   ELSE
       // ruch czarnych
       // 
       //ruch po skosie 
       #wykonuj_petle := TRUE;
       #poz_temp := #hetman.pozycja;
       WHILE #wykonuj_petle DO
           #poz_temp.x += 1;
           #poz_temp.y += 1;
           IF "sprawdz_czy_na_szachownicy"(#poz_temp) = true THEN
               IF "sprawdz_czy_wolne"(pozycja := #poz_temp, szachownica := #szachownica) = true THEN
                   IF #poz_temp.x = #polozenie_krola.x  AND #poz_temp.y = #polozenie_krola.y  THEN
                       #sprawdz_czy_hetman_szach := true;
                   END_IF;
               ELSIF "sprawdz_czy_zajete"(pozycja := #poz_temp, szachownica := #szachownica) = 2 THEN
                   IF #poz_temp.x = #polozenie_krola.x  AND #poz_temp.y = #polozenie_krola.y  THEN
                       #sprawdz_czy_hetman_szach := true;
                   ELSE
                       #wykonuj_petle := false;
                   END_IF;
               ELSE
                   #wykonuj_petle := false;
               END_IF;
           ELSE
               #wykonuj_petle := false;
           END_IF;
       END_WHILE;
       #wykonuj_petle := TRUE;
       #poz_temp := #hetman.pozycja;
       WHILE #wykonuj_petle DO
           #poz_temp.x += 1;
           #poz_temp.y -= 1;
           IF "sprawdz_czy_na_szachownicy"(#poz_temp) = true THEN
               IF "sprawdz_czy_wolne"(pozycja := #poz_temp, szachownica := #szachownica) = true THEN
                   IF #poz_temp.x = #polozenie_krola.x  AND #poz_temp.y = #polozenie_krola.y  THEN
                       #sprawdz_czy_hetman_szach := true;
                   END_IF;
               ELSIF "sprawdz_czy_zajete"(pozycja := #poz_temp, szachownica := #szachownica) = 2 THEN
                   IF #poz_temp.x = #polozenie_krola.x  AND #poz_temp.y = #polozenie_krola.y  THEN
                       #sprawdz_czy_hetman_szach := true;
                   ELSE
                       #wykonuj_petle := false;
                   END_IF;
               ELSE
                   #wykonuj_petle := false;
               END_IF;
           ELSE
               #wykonuj_petle := false;
           END_IF;
       END_WHILE;
       #wykonuj_petle := TRUE;
       #poz_temp := #hetman.pozycja;
       WHILE #wykonuj_petle DO
           #poz_temp.x -= 1;
           #poz_temp.y += 1;
           IF "sprawdz_czy_na_szachownicy"(#poz_temp) = true THEN
               IF "sprawdz_czy_wolne"(pozycja := #poz_temp, szachownica := #szachownica) = true THEN
                   IF #poz_temp.x = #polozenie_krola.x  AND #poz_temp.y = #polozenie_krola.y  THEN
                       #sprawdz_czy_hetman_szach := true;
                   END_IF;
               ELSIF "sprawdz_czy_zajete"(pozycja := #poz_temp, szachownica := #szachownica) = 2 THEN
                   IF #poz_temp.x = #polozenie_krola.x  AND #poz_temp.y = #polozenie_krola.y  THEN
                       #sprawdz_czy_hetman_szach := true;
                   ELSE
                       #wykonuj_petle := false;
                   END_IF;
               ELSE
                   #wykonuj_petle := false;
               END_IF;
           ELSE
               #wykonuj_petle := false;
           END_IF;
       END_WHILE;
       #wykonuj_petle := TRUE;
       #poz_temp := #hetman.pozycja;
       WHILE #wykonuj_petle DO
           #poz_temp.x -= 1;
           #poz_temp.y -= 1;
           IF "sprawdz_czy_na_szachownicy"(#poz_temp) = true THEN
               IF "sprawdz_czy_wolne"(pozycja := #poz_temp, szachownica := #szachownica) = true THEN
                   IF #poz_temp.x = #polozenie_krola.x  AND #poz_temp.y = #polozenie_krola.y  THEN
                       #sprawdz_czy_hetman_szach := true;
                   END_IF;
               ELSIF "sprawdz_czy_zajete"(pozycja := #poz_temp, szachownica := #szachownica) = 2 THEN
                   IF #poz_temp.x = #polozenie_krola.x  AND #poz_temp.y = #polozenie_krola.y  THEN
                       #sprawdz_czy_hetman_szach := true;
                   ELSE
                       #wykonuj_petle := false;
                   END_IF;
               ELSE
                   #wykonuj_petle := false;
               END_IF;
           ELSE
               #wykonuj_petle := false;
           END_IF;
       END_WHILE;
       //ruch poziomo i pionowo
       #wykonuj_petle := TRUE;
       #poz_temp := #hetman.pozycja;
       WHILE #wykonuj_petle DO
           #poz_temp.x += 1;
           #poz_temp.y += 0;
           IF "sprawdz_czy_na_szachownicy"(#poz_temp) = true THEN
               IF "sprawdz_czy_wolne"(pozycja := #poz_temp, szachownica := #szachownica) = true THEN
                   IF #poz_temp.x = #polozenie_krola.x  AND #poz_temp.y = #polozenie_krola.y  THEN
                       #sprawdz_czy_hetman_szach := true;
                   END_IF;
               ELSIF "sprawdz_czy_zajete"(pozycja := #poz_temp, szachownica := #szachownica) = 2 THEN
                   IF #poz_temp.x = #polozenie_krola.x  AND #poz_temp.y = #polozenie_krola.y  THEN
                       #sprawdz_czy_hetman_szach := true;
                   ELSE
                       #wykonuj_petle := false;
                   END_IF;
               ELSE
                   #wykonuj_petle := false;
               END_IF;
           ELSE
               #wykonuj_petle := false;
           END_IF;
       END_WHILE;
       #wykonuj_petle := TRUE;
       #poz_temp := #hetman.pozycja;
       WHILE #wykonuj_petle DO
           #poz_temp.x += 0;
           #poz_temp.y += 1;
           IF "sprawdz_czy_na_szachownicy"(#poz_temp) = true THEN
               IF "sprawdz_czy_wolne"(pozycja := #poz_temp, szachownica := #szachownica) = true THEN
                   IF #poz_temp.x = #polozenie_krola.x  AND #poz_temp.y = #polozenie_krola.y  THEN
                       #sprawdz_czy_hetman_szach := true;
                   END_IF;
               ELSIF "sprawdz_czy_zajete"(pozycja := #poz_temp, szachownica := #szachownica) = 2 THEN
                   IF #poz_temp.x = #polozenie_krola.x  AND #poz_temp.y = #polozenie_krola.y  THEN
                       #sprawdz_czy_hetman_szach := true;
                   ELSE
                       #wykonuj_petle := false;
                   END_IF;
               ELSE
                   #wykonuj_petle := false;
               END_IF;
           ELSE
               #wykonuj_petle := false;
           END_IF;
       END_WHILE;
       #wykonuj_petle := TRUE;
       #poz_temp := #hetman.pozycja;
       WHILE #wykonuj_petle DO
           #poz_temp.x += -1;
           #poz_temp.y += 0;
           IF "sprawdz_czy_na_szachownicy"(#poz_temp) = true THEN
               IF "sprawdz_czy_wolne"(pozycja := #poz_temp, szachownica := #szachownica) = true THEN
                   IF #poz_temp.x = #polozenie_krola.x  AND #poz_temp.y = #polozenie_krola.y  THEN
                       #sprawdz_czy_hetman_szach := true;
                   END_IF;
               ELSIF "sprawdz_czy_zajete"(pozycja := #poz_temp, szachownica := #szachownica) = 2 THEN
                   IF #poz_temp.x = #polozenie_krola.x  AND #poz_temp.y = #polozenie_krola.y  THEN
                       #sprawdz_czy_hetman_szach := true;
                   ELSE
                       #wykonuj_petle := false;
                   END_IF;
               ELSE
                   #wykonuj_petle := false;
               END_IF;
           ELSE
               #wykonuj_petle := false;
           END_IF;
       END_WHILE;
       #wykonuj_petle := TRUE;
       #poz_temp := #hetman.pozycja;
       WHILE #wykonuj_petle DO
           #poz_temp.x += 0;
           #poz_temp.y += -1;
           IF "sprawdz_czy_na_szachownicy"(#poz_temp) = true THEN
               IF "sprawdz_czy_wolne"(pozycja := #poz_temp, szachownica := #szachownica) = true THEN
                   IF #poz_temp.x = #polozenie_krola.x  AND #poz_temp.y = #polozenie_krola.y  THEN
                       #sprawdz_czy_hetman_szach := true;
                   END_IF;
               ELSIF "sprawdz_czy_zajete"(pozycja := #poz_temp, szachownica := #szachownica) = 2 THEN
                   IF #poz_temp.x = #polozenie_krola.x  AND #poz_temp.y = #polozenie_krola.y  THEN
                       #sprawdz_czy_hetman_szach := true;
                   ELSE
                       #wykonuj_petle := false;
                   END_IF;
               ELSE
                   #wykonuj_petle := false;
               END_IF;
           ELSE
               #wykonuj_petle := false;
           END_IF;
       END_WHILE;
   END_IF;
END_FUNCTION

// folder: wykrywanie_szach/Sprawdzanie ruchu figur

FUNCTION "Sprawdz_ruchy_figury_bez_sprawdzania" : Bool   // FC3, SCL
{ S7_Optimized_Access := 'TRUE' }
VERSION : 0.1
   VAR_INPUT
      szachownica : "Szachownica";
   END_VAR
   VAR_IN_OUT
      figura : "Figura";
   END_VAR
   VAR_TEMP
      pozycja_krola_bialego : "Pozycja";
      pozycja_krola_czarnego : "Pozycja";
      szach : Bool;
   END_VAR
BEGIN
   IF #figura.kolor = 1 THEN
       #pozycja_krola_czarnego := #szachownica.figury[28].pozycja;
       CASE #figura.rodzaj OF
           0:
              #szach :=  "sprawdz_czy_pion_szach"(szachownica := #szachownica,
                                                  polozenie_krola:=#pozycja_krola_czarnego, pion := #figura);
           1:
               #szach :=  "sprawdz_czy_goniec_szach"(szachownica := #szachownica,
                                          polozenie_krola:=#pozycja_krola_czarnego, goniec := #figura);
           2:
               #szach :=  "sprawdz_czy_skoczek_szach"(szachownica := #szachownica,
                                           polozenie_krola:=#pozycja_krola_czarnego, skoczek := #figura);
           3:
               #szach :=  "sprawdz_czy_wieza_szach"(szachownica := #szachownica,
                                         polozenie_krola:=#pozycja_krola_czarnego, wieza := #figura);
           4:
               #szach := "sprawdz_czy_hetman_szach"(szachownica := #szachownica,
                                          polozenie_krola:=#pozycja_krola_czarnego, hetman := #figura);
           5:
               #szach :=  "sprawdz_czy_krol_szach"(szachownica := #szachownica,
                                        polozenie_krola:=#pozycja_krola_czarnego, krol := #figura);

           ELSE
               ;
       END_CASE;
   ELSE

       #pozycja_krola_bialego := #szachownica.figury[4].pozycja;
       CASE #figura.rodzaj OF
           0:
               #szach := "sprawdz_czy_pion_szach"(szachownica := #szachownica,
                                                  polozenie_krola := #pozycja_krola_bialego, pion := #figura);
           1:
               #szach := "sprawdz_czy_goniec_szach"(szachownica := #szachownica,
                                                    polozenie_krola := #pozycja_krola_bialego, goniec := #figura);
           2:
               #szach := "sprawdz_czy_skoczek_szach"(szachownica := #szachownica,
                                                     polozenie_krola := #pozycja_krola_bialego, skoczek := #figura);
           3:
               #szach := "sprawdz_czy_wieza_szach"(szachownica := #szachownica,
                                                   polozenie_krola := #pozycja_krola_bialego, wieza := #figura);
           4:
               #szach := "sprawdz_czy_hetman_szach"(szachownica := #szachownica,
                                                    polozenie_krola := #pozycja_krola_bialego, hetman := #figura);
           5:
               #szach := "sprawdz_czy_krol_szach"(szachownica := #szachownica,
                                                  polozenie_krola := #pozycja_krola_bialego, krol := #figura);

           ELSE
               ;
       END_CASE;
   END_IF;
   #Sprawdz_ruchy_figury_bez_sprawdzania := #szach;
END_FUNCTION

FUNCTION "Wykrywanie_ruchów" : Int   // FC5, SCL
{ S7_Optimized_Access := 'TRUE' }
VERSION : 0.1
   VAR_INPUT
      tura_bool : Bool;
   END_VAR
   VAR_IN_OUT
      Szachownica : "Szachownica";
   END_VAR
   VAR_TEMP
      i : Int;
      licznik_ruchow : Int;
   END_VAR
BEGIN
   #licznik_ruchow := 0;
   IF #tura_bool THEN
       FOR #i := 0 TO 15 DO
           IF #Szachownica.figury[#i].zywy = 1 THEN
               #licznik_ruchow +=  "Sprawdz_ruchy_figury_ze_sprawdzaniem"(figura := #Szachownica.figury[#i],
                                                      szachownica := "Status_rozgrywki".Szachownica);
           END_IF;
       END_FOR;
   ELSE
       FOR #i := 16 TO 31 DO
           IF #Szachownica.figury[#i].zywy = 1 THEN
               #licznik_ruchow += "Sprawdz_ruchy_figury_ze_sprawdzaniem"(figura := #Szachownica.figury[#i],
                                                                         szachownica := "Status_rozgrywki".Szachownica);
           END_IF;
       END_FOR;
   END_IF;

   #Wykrywanie_ruchów := #licznik_ruchow;
END_FUNCTION

FUNCTION "Sprawdz_ruchy_figury_ze_sprawdzaniem" : Int   // FC6, SCL
{ S7_Optimized_Access := 'TRUE' }
VERSION : 0.1
   VAR_INPUT
      szachownica : "Szachownica";
   END_VAR
   VAR_IN_OUT
      figura : "Figura";
   END_VAR
   VAR_TEMP
      licznik_ruchow : Int;
   END_VAR
BEGIN
   CASE #figura.rodzaj OF
       0:
           #licznik_ruchow:= "sprawdz_ruch_piona"(szachownica := #szachownica,
                                pion := #figura);
       1:
           #licznik_ruchow:="sprawdz_ruch_gońca"(szachownica := #szachownica,
                                goniec := #figura);
       2:
           #licznik_ruchow:= "sprawdz_ruch_skoczka"(szachownica := #szachownica,
                                  skoczek := #figura);
       3:
           #licznik_ruchow:= "sprawdz_ruch_wieży"(szachownica := #szachownica,
                                wieza := #figura);
       4:
           #licznik_ruchow:= "sprawdz_ruch_hetmana"(szachownica := #szachownica,
                                  hetman := #figura);
       5:
           #licznik_ruchow:="sprawdz_ruch_króla"(szachownica := #szachownica,
                                krol := #figura);

       ELSE  // Statement section ELSE
           ;
   END_CASE;
   #Sprawdz_ruchy_figury_ze_sprawdzaniem := #licznik_ruchow;
END_FUNCTION

FUNCTION "sprawdz_ruch_piona" : Int   // FC7, SCL
{ S7_Optimized_Access := 'TRUE' }
VERSION : 0.1
   VAR_INPUT
      szachownica : "Szachownica";
   END_VAR
   VAR_IN_OUT
      pion : "Figura";
   END_VAR
   VAR_TEMP
      poz_temp : "Pozycja";
      indeks_mozliwych_ruchow : Int;
      fig_temp : "Figura";
   END_VAR
BEGIN
   #indeks_mozliwych_ruchow := 0;
   IF #pion.kolor = 1 THEN
       IF #pion.pozycja.y = 2 THEN
           #poz_temp := #pion.pozycja;
           #poz_temp.x := #pion.pozycja.x;
           #poz_temp.y := #pion.pozycja.y + 2;
           IF "sprawdz_czy_na_szachownicy"(#poz_temp) THEN
               IF "sprawdz_czy_wolne"(pozycja := #poz_temp, szachownica := #szachownica) = 1 THEN
                   IF "sprawdz_czy_ruch_możliwy"(figura := #pion, szachownica := #szachownica, pozycja := #poz_temp) = true THEN
                       #pion.mozliwe_ruchy[#indeks_mozliwych_ruchow] := #poz_temp;
                       #indeks_mozliwych_ruchow += 1;
                   END_IF;
               END_IF;
           END_IF;
       END_IF;
       #poz_temp.x := #pion.pozycja.x;
       #poz_temp.y := #pion.pozycja.y + 1;
       IF "sprawdz_czy_na_szachownicy"(#poz_temp) THEN
           IF "sprawdz_czy_wolne"(pozycja := #poz_temp, szachownica := #szachownica) = 1 THEN
               IF "sprawdz_czy_ruch_możliwy"(figura := #pion, szachownica := #szachownica, pozycja := #poz_temp) = true THEN
                   #pion.mozliwe_ruchy[#indeks_mozliwych_ruchow] := #poz_temp;
                   #indeks_mozliwych_ruchow += 1;
               END_IF;
           END_IF;
       END_IF;
       #poz_temp.x := #pion.pozycja.x - 1;
       #poz_temp.y := #pion.pozycja.y + 1;
       IF "sprawdz_czy_na_szachownicy"(#poz_temp) THEN
           IF "sprawdz_czy_zajete"(pozycja := #poz_temp, szachownica := #szachownica) = 1 THEN
               IF "sprawdz_czy_ruch_możliwy"(figura := #pion, szachownica := #szachownica, pozycja := #poz_temp) = true THEN
                   #pion.mozliwe_ruchy[#indeks_mozliwych_ruchow] := #poz_temp;
                   #indeks_mozliwych_ruchow += 1;
               END_IF;
           END_IF;
       END_IF;
       #poz_temp.x := #pion.pozycja.x + 1;
       #poz_temp.y := #pion.pozycja.y + 1;
       IF "sprawdz_czy_na_szachownicy"(#poz_temp) THEN
           IF "sprawdz_czy_zajete"(pozycja := #poz_temp, szachownica := #szachownica) = 1 THEN
               IF "sprawdz_czy_ruch_możliwy"(figura := #pion, szachownica := #szachownica, pozycja := #poz_temp) = true THEN
                   #pion.mozliwe_ruchy[#indeks_mozliwych_ruchow] := #poz_temp;
                   #indeks_mozliwych_ruchow += 1;
               END_IF;
           END_IF;
       END_IF;
       //bicie w przelocie 
       #poz_temp.x := #pion.pozycja.x + 1;
       #poz_temp.y := #pion.pozycja.y;
       IF "sprawdz_czy_na_szachownicy"(#poz_temp) THEN
           IF "sprawdz_czy_zajete"(pozycja := #poz_temp, szachownica := #szachownica) = 1 AND
               "konwersja_pozycja_na_figura"(pozycja := #poz_temp, Szachownica := #szachownica, figura => #fig_temp) THEN
               IF #fig_temp.tura_1_ruchu_piona = "Status_rozgrywki".tura_int -1 THEN
                   #poz_temp.x := #pion.pozycja.x + 1;
                   #poz_temp.y := #pion.pozycja.y + 1;
                   IF "sprawdz_czy_wolne"(szachownica := #szachownica, pozycja := #poz_temp) THEN
                       IF "sprawdz_czy_ruch_możliwy"(figura := #pion, szachownica := #szachownica, pozycja := #poz_temp) = true THEN
                           #pion.mozliwe_ruchy[#indeks_mozliwych_ruchow] := #poz_temp;
                           #indeks_mozliwych_ruchow += 1;
                       END_IF;
                   END_IF;
               END_IF;
           END_IF;
       END_IF;
       #poz_temp.x := #pion.pozycja.x - 1;
       #poz_temp.y := #pion.pozycja.y;
       IF "sprawdz_czy_na_szachownicy"(#poz_temp) THEN
           IF "sprawdz_czy_zajete"(pozycja := #poz_temp, szachownica := #szachownica) = 1 AND
               "konwersja_pozycja_na_figura"(pozycja := #poz_temp, Szachownica := #szachownica, figura => #fig_temp) THEN
               IF #fig_temp.tura_1_ruchu_piona = "Status_rozgrywki".tura_int - 1 THEN
                   #poz_temp.x := #pion.pozycja.x - 1;
                   #poz_temp.y := #pion.pozycja.y + 1;
                   IF "sprawdz_czy_wolne"(szachownica := #szachownica, pozycja := #poz_temp) THEN
                       IF "sprawdz_czy_ruch_możliwy"(figura := #pion, szachownica := #szachownica, pozycja := #poz_temp) = true THEN
                           #pion.mozliwe_ruchy[#indeks_mozliwych_ruchow] := #poz_temp;
                           #indeks_mozliwych_ruchow += 1;
                       END_IF;
                   END_IF;
               END_IF;
            END_IF;
         END_IF;
   ELSE
       IF #pion.pozycja.y = 7 THEN
           #poz_temp.x := #pion.pozycja.x;
           #poz_temp.y := #pion.pozycja.y - 2;
           IF "sprawdz_czy_na_szachownicy"(#poz_temp) THEN
               IF "sprawdz_czy_wolne"(pozycja := #poz_temp, szachownica := #szachownica) = 1 THEN
                   IF "sprawdz_czy_ruch_możliwy"(figura := #pion, szachownica := #szachownica, pozycja := #poz_temp) = true THEN
                       #pion.mozliwe_ruchy[#indeks_mozliwych_ruchow] := #poz_temp;
                       #indeks_mozliwych_ruchow += 1;
                   END_IF;
               END_IF;
           END_IF;
       END_IF;
       #poz_temp.x := #pion.pozycja.x;
       #poz_temp.y := #pion.pozycja.y - 1;
       IF "sprawdz_czy_na_szachownicy"(#poz_temp) THEN
           IF "sprawdz_czy_wolne"(pozycja := #poz_temp, szachownica := #szachownica) = 1 THEN
               IF "sprawdz_czy_ruch_możliwy"(figura := #pion, szachownica := #szachownica, pozycja := #poz_temp) = true THEN
                   #pion.mozliwe_ruchy[#indeks_mozliwych_ruchow] := #poz_temp;
                   #indeks_mozliwych_ruchow += 1;
               END_IF;
           END_IF;
       END_IF;
       #poz_temp.x := #pion.pozycja.x - 1;
       #poz_temp.y := #pion.pozycja.y - 1;
       IF "sprawdz_czy_na_szachownicy"(#poz_temp) THEN
           IF "sprawdz_czy_zajete"(pozycja := #poz_temp, szachownica := #szachownica) = 2 THEN
               IF "sprawdz_czy_ruch_możliwy"(figura := #pion, szachownica := #szachownica, pozycja := #poz_temp) = true THEN
                   #pion.mozliwe_ruchy[#indeks_mozliwych_ruchow] := #poz_temp;
                   #indeks_mozliwych_ruchow += 1;
               END_IF;
           END_IF;
       END_IF;
       #poz_temp.x := #pion.pozycja.x + 1;
       #poz_temp.y := #pion.pozycja.y - 1;
       IF "sprawdz_czy_na_szachownicy"(#poz_temp) THEN
           IF "sprawdz_czy_zajete"(pozycja := #poz_temp, szachownica := #szachownica) = 2 THEN
               IF "sprawdz_czy_ruch_możliwy"(figura := #pion, szachownica := #szachownica, pozycja := #poz_temp) = true THEN
                   #pion.mozliwe_ruchy[#indeks_mozliwych_ruchow] := #poz_temp;
                   #indeks_mozliwych_ruchow += 1;
               END_IF;
           END_IF;
       END_IF;
       //bicie w przelocie 
       #poz_temp.x := #pion.pozycja.x + 1;
       #poz_temp.y := #pion.pozycja.y;
       IF "sprawdz_czy_na_szachownicy"(#poz_temp) THEN
           IF "sprawdz_czy_zajete"(pozycja := #poz_temp, szachownica := #szachownica) = 2 AND
               "konwersja_pozycja_na_figura"(pozycja := #poz_temp, Szachownica := #szachownica, figura => #fig_temp) THEN
               IF #fig_temp.tura_1_ruchu_piona = "Status_rozgrywki".tura_int - 1 THEN
                   #poz_temp.x := #pion.pozycja.x + 1;
                   #poz_temp.y := #pion.pozycja.y + 1;
                   IF "sprawdz_czy_wolne"(szachownica := #szachownica, pozycja := #poz_temp) THEN
                       IF "sprawdz_czy_ruch_możliwy"(figura := #pion, szachownica := #szachownica, pozycja := #poz_temp) = true THEN
                           #pion.mozliwe_ruchy[#indeks_mozliwych_ruchow] := #poz_temp;
                           #indeks_mozliwych_ruchow += 1;
                       END_IF;
                   END_IF;
               END_IF;
           END_IF;
       END_IF;
       #poz_temp.x := #pion.pozycja.x - 1;
       #poz_temp.y := #pion.pozycja.y;
       IF "sprawdz_czy_na_szachownicy"(#poz_temp) THEN
           IF "sprawdz_czy_zajete"(pozycja := #poz_temp, szachownica := #szachownica) = 2 AND
               "konwersja_pozycja_na_figura"(pozycja := #poz_temp, Szachownica := #szachownica, figura => #fig_temp) THEN
               IF #fig_temp.tura_1_ruchu_piona = "Status_rozgrywki".tura_int - 1 THEN
                   #poz_temp.x := #pion.pozycja.x - 1;
                   #poz_temp.y := #pion.pozycja.y + 1;
                   IF "sprawdz_czy_wolne"(szachownica := #szachownica, pozycja := #poz_temp) THEN
                       IF "sprawdz_czy_ruch_możliwy"(figura := #pion, szachownica := #szachownica, pozycja := #poz_temp) = true THEN
                           #pion.mozliwe_ruchy[#indeks_mozliwych_ruchow] := #poz_temp;
                           #indeks_mozliwych_ruchow += 1;
                       END_IF;
                   END_IF;
               END_IF;
           END_IF;
       END_IF;
   END_IF;
       #sprawdz_ruch_piona := #indeks_mozliwych_ruchow;
END_FUNCTION

FUNCTION "sprawdz_czy_wolne" : Bool   // FC8, SCL
{ S7_Optimized_Access := 'TRUE' }
VERSION : 0.1
   VAR_INPUT
      pozycja : "Pozycja";   // pozycja do sprawdzenia
      szachownica : "Szachownica";
   END_VAR
   VAR_TEMP
      i : Int;
   END_VAR
BEGIN
   #sprawdz_czy_wolne := true;
       FOR #i := 0 TO 31 DO
           IF #szachownica.figury[#i].pozycja.x = #pozycja.x AND
               #szachownica.figury[#i].pozycja.y = #pozycja.y THEN
               #sprawdz_czy_wolne := false;
           END_IF;
       END_FOR;
END_FUNCTION

FUNCTION "sprawdz_czy_zajete" : Int   // FC9, SCL
{ S7_Optimized_Access := 'TRUE' }
VERSION : 0.1
   VAR_INPUT
      pozycja : "Pozycja";   // pozycja do sprawdzenia
      szachownica : "Szachownica";
   END_VAR
   VAR_TEMP
      i : Int;
   END_VAR
BEGIN

   #sprawdz_czy_zajete := 0;
       FOR #i := 0 TO 31 DO
           IF #szachownica.figury[#i].pozycja.x = #pozycja.x AND
               #szachownica.figury[#i].pozycja.y = #pozycja.y THEN
               IF #szachownica.figury[#i].kolor = 0 THEN
                   #sprawdz_czy_zajete := 1;
               ELSE
                   #sprawdz_czy_zajete := 2;
               END_IF;
           END_IF;
       END_FOR;
END_FUNCTION

FUNCTION "sprawdz_ruch_skoczka" : Int   // FC10, SCL
{ S7_Optimized_Access := 'TRUE' }
VERSION : 0.1
   VAR_INPUT
      szachownica : "Szachownica";
   END_VAR
   VAR_IN_OUT
      skoczek : "Figura";
   END_VAR
   VAR_TEMP
      poz_temp : "Pozycja";
      indeks_mozliwych_ruchow : Int;
   END_VAR
BEGIN
   #indeks_mozliwych_ruchow := 0;
   IF #skoczek.kolor = 1 THEN
       // ruchy skoczka bialego we wszystkich kierunkach
       #poz_temp := #skoczek.pozycja;
       #poz_temp.x := #skoczek.pozycja.x + 2;
       #poz_temp.y := #skoczek.pozycja.y + 1;
       IF "sprawdz_czy_na_szachownicy"(#poz_temp) = true THEN
           IF "sprawdz_czy_wolne"(pozycja := #poz_temp, szachownica := #szachownica) = true THEN
               IF "sprawdz_czy_ruch_możliwy"(figura := #skoczek, szachownica := #szachownica, pozycja := #poz_temp)  = true THEN
                   #skoczek.mozliwe_ruchy[#indeks_mozliwych_ruchow] := #poz_temp;
                   #indeks_mozliwych_ruchow += 1;
               END_IF;
           ELSIF "sprawdz_czy_zajete"(pozycja := #poz_temp, szachownica := #szachownica) = 1 THEN
               IF "sprawdz_czy_ruch_możliwy"(figura := #skoczek, szachownica := #szachownica, pozycja := #poz_temp)  = true THEN
                   #skoczek.mozliwe_ruchy[#indeks_mozliwych_ruchow] := #poz_temp;
                   #indeks_mozliwych_ruchow += 1;
               END_IF;
           END_IF;
       END_IF;
       #poz_temp := #skoczek.pozycja;
       #poz_temp.x := #skoczek.pozycja.x + 2;
       #poz_temp.y := #skoczek.pozycja.y - 1;
       IF "sprawdz_czy_na_szachownicy"(#poz_temp) = true THEN
           IF "sprawdz_czy_wolne"(pozycja := #poz_temp, szachownica := #szachownica) = true THEN
               IF "sprawdz_czy_ruch_możliwy"(figura := #skoczek, szachownica := #szachownica, pozycja := #poz_temp)  = true THEN
                   #skoczek.mozliwe_ruchy[#indeks_mozliwych_ruchow] := #poz_temp;
                   #indeks_mozliwych_ruchow += 1;
               END_IF;
           ELSIF "sprawdz_czy_zajete"(pozycja := #poz_temp, szachownica := #szachownica) = 1 THEN
               IF "sprawdz_czy_ruch_możliwy"(figura := #skoczek, szachownica := #szachownica, pozycja := #poz_temp)  = true THEN
                   #skoczek.mozliwe_ruchy[#indeks_mozliwych_ruchow] := #poz_temp;
                   #indeks_mozliwych_ruchow += 1;
               END_IF;
           END_IF;
       END_IF;
       #poz_temp := #skoczek.pozycja;
       #poz_temp.x := #skoczek.pozycja.x - 2;
       #poz_temp.y := #skoczek.pozycja.y + 1;
       IF "sprawdz_czy_na_szachownicy"(#poz_temp) = true THEN
           IF "sprawdz_czy_wolne"(pozycja := #poz_temp, szachownica := #szachownica) = true THEN
               IF "sprawdz_czy_ruch_możliwy"(figura := #skoczek, szachownica := #szachownica, pozycja := #poz_temp)  = true THEN
                   #skoczek.mozliwe_ruchy[#indeks_mozliwych_ruchow] := #poz_temp;
                   #indeks_mozliwych_ruchow += 1;
               END_IF;
           ELSIF "sprawdz_czy_zajete"(pozycja := #poz_temp, szachownica := #szachownica) = 1 THEN
               IF "sprawdz_czy_ruch_możliwy"(figura := #skoczek, szachownica := #szachownica, pozycja := #poz_temp)  = true THEN
                   #skoczek.mozliwe_ruchy[#indeks_mozliwych_ruchow] := #poz_temp;
                   #indeks_mozliwych_ruchow += 1;
               END_IF;
           END_IF;
       END_IF;
       #poz_temp := #skoczek.pozycja;
       #poz_temp.x := #skoczek.pozycja.x - 2;
       #poz_temp.y := #skoczek.pozycja.y - 1;
       IF "sprawdz_czy_na_szachownicy"(#poz_temp) = true THEN
           IF "sprawdz_czy_wolne"(pozycja := #poz_temp, szachownica := #szachownica) = true THEN
               IF "sprawdz_czy_ruch_możliwy"(figura := #skoczek, szachownica := #szachownica, pozycja := #poz_temp)  = true THEN
                   #skoczek.mozliwe_ruchy[#indeks_mozliwych_ruchow] := #poz_temp;
                   #indeks_mozliwych_ruchow += 1;
               END_IF;
           ELSIF "sprawdz_czy_zajete"(pozycja := #poz_temp, szachownica := #szachownica) = 1 THEN
               IF "sprawdz_czy_ruch_możliwy"(figura := #skoczek, szachownica := #szachownica, pozycja := #poz_temp)  = true THEN
                   #skoczek.mozliwe_ruchy[#indeks_mozliwych_ruchow] := #poz_temp;
                   #indeks_mozliwych_ruchow += 1;
               END_IF;
           END_IF;
       END_IF;
       #poz_temp := #skoczek.pozycja;
       #poz_temp.x := #skoczek.pozycja.x + 1;
       #poz_temp.y := #skoczek.pozycja.y + 2;
       IF "sprawdz_czy_na_szachownicy"(#poz_temp) = true THEN
           IF "sprawdz_czy_wolne"(pozycja := #poz_temp, szachownica := #szachownica) = true THEN
               IF "sprawdz_czy_ruch_możliwy"(figura := #skoczek, szachownica := #szachownica, pozycja := #poz_temp)  = true THEN
                   #skoczek.mozliwe_ruchy[#indeks_mozliwych_ruchow] := #poz_temp;
                   #indeks_mozliwych_ruchow += 1;
               END_IF;
           ELSIF "sprawdz_czy_zajete"(pozycja := #poz_temp, szachownica := #szachownica) = 1 THEN
               IF "sprawdz_czy_ruch_możliwy"(figura := #skoczek, szachownica := #szachownica, pozycja := #poz_temp)  = true THEN
                   #skoczek.mozliwe_ruchy[#indeks_mozliwych_ruchow] := #poz_temp;
                   #indeks_mozliwych_ruchow += 1;
               END_IF;
           END_IF;
       END_IF;
       #poz_temp := #skoczek.pozycja;
       #poz_temp.x := #skoczek.pozycja.x - 1;
       #poz_temp.y := #skoczek.pozycja.y + 2;
       IF "sprawdz_czy_na_szachownicy"(#poz_temp) = true THEN
           IF "sprawdz_czy_wolne"(pozycja := #poz_temp, szachownica := #szachownica) = true THEN
               IF "sprawdz_czy_ruch_możliwy"(figura := #skoczek, szachownica := #szachownica, pozycja := #poz_temp)  = true THEN
                   #skoczek.mozliwe_ruchy[#indeks_mozliwych_ruchow] := #poz_temp;
                   #indeks_mozliwych_ruchow += 1;
               END_IF;
           ELSIF "sprawdz_czy_zajete"(pozycja := #poz_temp, szachownica := #szachownica) = 1 THEN
               IF "sprawdz_czy_ruch_możliwy"(figura := #skoczek, szachownica := #szachownica, pozycja := #poz_temp)  = true THEN
                   #skoczek.mozliwe_ruchy[#indeks_mozliwych_ruchow] := #poz_temp;
                   #indeks_mozliwych_ruchow += 1;
               END_IF;
           END_IF;
       END_IF;
       #poz_temp := #skoczek.pozycja;
       #poz_temp.x := #skoczek.pozycja.x + 1;
       #poz_temp.y := #skoczek.pozycja.y - 2;
       IF "sprawdz_czy_na_szachownicy"(#poz_temp) = true THEN
           IF "sprawdz_czy_wolne"(pozycja := #poz_temp, szachownica := #szachownica) = true THEN
               IF "sprawdz_czy_ruch_możliwy"(figura := #skoczek, szachownica := #szachownica, pozycja := #poz_temp)  = true THEN
                   #skoczek.mozliwe_ruchy[#indeks_mozliwych_ruchow] := #poz_temp;
                   #indeks_mozliwych_ruchow += 1;
               END_IF;
           ELSIF "sprawdz_czy_zajete"(pozycja := #poz_temp, szachownica := #szachownica) = 1 THEN
               IF "sprawdz_czy_ruch_możliwy"(figura := #skoczek, szachownica := #szachownica, pozycja := #poz_temp)  = true THEN
                   #skoczek.mozliwe_ruchy[#indeks_mozliwych_ruchow] := #poz_temp;
                   #indeks_mozliwych_ruchow += 1;
               END_IF;
           END_IF;
       END_IF;
       #poz_temp := #skoczek.pozycja;
       #poz_temp.x := #skoczek.pozycja.x - 1;
       #poz_temp.y := #skoczek.pozycja.y - 2;
       IF "sprawdz_czy_na_szachownicy"(#poz_temp) = true THEN
           IF "sprawdz_czy_wolne"(pozycja := #poz_temp, szachownica := #szachownica) = true THEN
               IF "sprawdz_czy_ruch_możliwy"(figura := #skoczek, szachownica := #szachownica, pozycja := #poz_temp)  = true THEN
                   #skoczek.mozliwe_ruchy[#indeks_mozliwych_ruchow] := #poz_temp;
                   #indeks_mozliwych_ruchow += 1;
               END_IF;
           ELSIF "sprawdz_czy_zajete"(pozycja := #poz_temp, szachownica := #szachownica) = 1 THEN
               IF "sprawdz_czy_ruch_możliwy"(figura := #skoczek, szachownica := #szachownica, pozycja := #poz_temp)  = true THEN
                   #skoczek.mozliwe_ruchy[#indeks_mozliwych_ruchow] := #poz_temp;
                   #indeks_mozliwych_ruchow += 1;
               END_IF;
           END_IF;
       END_IF;




   ELSE
       // ruchy skoczka czarnego we wszystkich kierunkach
       #poz_temp := #skoczek.pozycja;
       #poz_temp.x := #skoczek.pozycja.x + 2;
       #poz_temp.y := #skoczek.pozycja.y + 1;
       IF "sprawdz_czy_na_szachownicy"(#poz_temp) = true THEN
           IF "sprawdz_czy_wolne"(pozycja := #poz_temp, szachownica := #szachownica) = true THEN
               IF "sprawdz_czy_ruch_możliwy"(figura := #skoczek, szachownica := #szachownica, pozycja := #poz_temp)  = true THEN
                   #skoczek.mozliwe_ruchy[#indeks_mozliwych_ruchow] := #poz_temp;
                   #indeks_mozliwych_ruchow += 1;
               END_IF;
           ELSIF "sprawdz_czy_zajete"(pozycja := #poz_temp, szachownica := #szachownica) = 2 THEN
               IF "sprawdz_czy_ruch_możliwy"(figura := #skoczek, szachownica := #szachownica, pozycja := #poz_temp)  = true THEN
                   #skoczek.mozliwe_ruchy[#indeks_mozliwych_ruchow] := #poz_temp;
                   #indeks_mozliwych_ruchow += 1;
               END_IF;
           END_IF;
       END_IF;
       #poz_temp := #skoczek.pozycja;
       #poz_temp.x := #skoczek.pozycja.x + 2;
       #poz_temp.y := #skoczek.pozycja.y - 1;
       IF "sprawdz_czy_na_szachownicy"(#poz_temp) = true THEN
           IF "sprawdz_czy_wolne"(pozycja := #poz_temp, szachownica := #szachownica) = true THEN
               IF "sprawdz_czy_ruch_możliwy"(figura := #skoczek, szachownica := #szachownica, pozycja := #poz_temp)  = true THEN
                   #skoczek.mozliwe_ruchy[#indeks_mozliwych_ruchow] := #poz_temp;
                   #indeks_mozliwych_ruchow += 1;
               END_IF;
           ELSIF "sprawdz_czy_zajete"(pozycja := #poz_temp, szachownica := #szachownica) = 2 THEN
               IF "sprawdz_czy_ruch_możliwy"(figura := #skoczek, szachownica := #szachownica, pozycja := #poz_temp)  = true THEN
                   #skoczek.mozliwe_ruchy[#indeks_mozliwych_ruchow] := #poz_temp;
                   #indeks_mozliwych_ruchow += 1;
               END_IF;
           END_IF;
       END_IF;
       #poz_temp := #skoczek.pozycja;
       #poz_temp.x := #skoczek.pozycja.x - 2;
       #poz_temp.y := #skoczek.pozycja.y + 1;
       IF "sprawdz_czy_na_szachownicy"(#poz_temp) = true THEN
           IF "sprawdz_czy_wolne"(pozycja := #poz_temp, szachownica := #szachownica) = true THEN
               IF "sprawdz_czy_ruch_możliwy"(figura := #skoczek, szachownica := #szachownica, pozycja := #poz_temp)  = true THEN
                   #skoczek.mozliwe_ruchy[#indeks_mozliwych_ruchow] := #poz_temp;
                   #indeks_mozliwych_ruchow += 1;
               END_IF;
           ELSIF "sprawdz_czy_zajete"(pozycja := #poz_temp, szachownica := #szachownica) = 2 THEN
               IF "sprawdz_czy_ruch_możliwy"(figura := #skoczek, szachownica := #szachownica, pozycja := #poz_temp)  = true THEN
                   #skoczek.mozliwe_ruchy[#indeks_mozliwych_ruchow] := #poz_temp;
                   #indeks_mozliwych_ruchow += 1;
               END_IF;
           END_IF;
       END_IF;
       #poz_temp := #skoczek.pozycja;
       #poz_temp.x := #skoczek.pozycja.x - 2;
       #poz_temp.y := #skoczek.pozycja.y - 1;
       IF "sprawdz_czy_na_szachownicy"(#poz_temp) = true THEN
           IF "sprawdz_czy_wolne"(pozycja := #poz_temp, szachownica := #szachownica) = true THEN
               IF "sprawdz_czy_ruch_możliwy"(figura := #skoczek, szachownica := #szachownica, pozycja := #poz_temp)  = true THEN
                   #skoczek.mozliwe_ruchy[#indeks_mozliwych_ruchow] := #poz_temp;
                   #indeks_mozliwych_ruchow += 1;
               END_IF;
           ELSIF "sprawdz_czy_zajete"(pozycja := #poz_temp, szachownica := #szachownica) = 2 THEN
               IF "sprawdz_czy_ruch_możliwy"(figura := #skoczek, szachownica := #szachownica, pozycja := #poz_temp)  = true THEN
                   #skoczek.mozliwe_ruchy[#indeks_mozliwych_ruchow] := #poz_temp;
                   #indeks_mozliwych_ruchow += 1;
               END_IF;
           END_IF;
       END_IF;
       #poz_temp := #skoczek.pozycja;
       #poz_temp.x := #skoczek.pozycja.x + 1;
       #poz_temp.y := #skoczek.pozycja.y + 2;
       IF "sprawdz_czy_na_szachownicy"(#poz_temp) = true THEN
           IF "sprawdz_czy_wolne"(pozycja := #poz_temp, szachownica := #szachownica) = true THEN
               IF "sprawdz_czy_ruch_możliwy"(figura := #skoczek, szachownica := #szachownica, pozycja := #poz_temp)  = true THEN
                   #skoczek.mozliwe_ruchy[#indeks_mozliwych_ruchow] := #poz_temp;
                   #indeks_mozliwych_ruchow += 1;
               END_IF;
           ELSIF "sprawdz_czy_zajete"(pozycja := #poz_temp, szachownica := #szachownica) = 2 THEN
               IF "sprawdz_czy_ruch_możliwy"(figura := #skoczek, szachownica := #szachownica, pozycja := #poz_temp)  = true THEN
                   #skoczek.mozliwe_ruchy[#indeks_mozliwych_ruchow] := #poz_temp;
                   #indeks_mozliwych_ruchow += 1;
               END_IF;
           END_IF;
       END_IF;
       #poz_temp := #skoczek.pozycja;
       #poz_temp.x := #skoczek.pozycja.x - 1;
       #poz_temp.y := #skoczek.pozycja.y + 2;
       IF "sprawdz_czy_na_szachownicy"(#poz_temp) = true THEN
           IF "sprawdz_czy_wolne"(pozycja := #poz_temp, szachownica := #szachownica) = true THEN
               IF "sprawdz_czy_ruch_możliwy"(figura := #skoczek, szachownica := #szachownica, pozycja := #poz_temp)  = true THEN
                   #skoczek.mozliwe_ruchy[#indeks_mozliwych_ruchow] := #poz_temp;
                   #indeks_mozliwych_ruchow += 1;
               END_IF;
           ELSIF "sprawdz_czy_zajete"(pozycja := #poz_temp, szachownica := #szachownica) = 2 THEN
               IF "sprawdz_czy_ruch_możliwy"(figura := #skoczek, szachownica := #szachownica, pozycja := #poz_temp)  = true THEN
                   #skoczek.mozliwe_ruchy[#indeks_mozliwych_ruchow] := #poz_temp;
                   #indeks_mozliwych_ruchow += 1;
               END_IF;
           END_IF;
       END_IF;
       #poz_temp := #skoczek.pozycja;
       #poz_temp.x := #skoczek.pozycja.x + 1;
       #poz_temp.y := #skoczek.pozycja.y - 2;
       IF "sprawdz_czy_na_szachownicy"(#poz_temp) = true THEN
           IF "sprawdz_czy_wolne"(pozycja := #poz_temp, szachownica := #szachownica) = true THEN
               IF "sprawdz_czy_ruch_możliwy"(figura := #skoczek, szachownica := #szachownica, pozycja := #poz_temp)  = true THEN
                   #skoczek.mozliwe_ruchy[#indeks_mozliwych_ruchow] := #poz_temp;
                   #indeks_mozliwych_ruchow += 1;
               END_IF;
           ELSIF "sprawdz_czy_zajete"(pozycja := #poz_temp, szachownica := #szachownica) = 2 THEN
               IF "sprawdz_czy_ruch_możliwy"(figura := #skoczek, szachownica := #szachownica, pozycja := #poz_temp)  = true THEN
                   #skoczek.mozliwe_ruchy[#indeks_mozliwych_ruchow] := #poz_temp;
                   #indeks_mozliwych_ruchow += 1;
               END_IF;
           END_IF;
       END_IF;
       #poz_temp := #skoczek.pozycja;
       #poz_temp.x := #skoczek.pozycja.x - 1;
       #poz_temp.y := #skoczek.pozycja.y - 2;
       IF "sprawdz_czy_na_szachownicy"(#poz_temp) = true THEN
           IF "sprawdz_czy_wolne"(pozycja := #poz_temp, szachownica := #szachownica) = true THEN
               IF "sprawdz_czy_ruch_możliwy"(figura := #skoczek, szachownica := #szachownica, pozycja := #poz_temp)  = true THEN
                   #skoczek.mozliwe_ruchy[#indeks_mozliwych_ruchow] := #poz_temp;
                   #indeks_mozliwych_ruchow += 1;
               END_IF;
           ELSIF "sprawdz_czy_zajete"(pozycja := #poz_temp, szachownica := #szachownica) = 2 THEN
               IF "sprawdz_czy_ruch_możliwy"(figura := #skoczek, szachownica := #szachownica, pozycja := #poz_temp)  = true THEN
                   #skoczek.mozliwe_ruchy[#indeks_mozliwych_ruchow] := #poz_temp;
                   #indeks_mozliwych_ruchow += 1;
               END_IF;
           END_IF;
       END_IF;

   END_IF;
   #sprawdz_ruch_skoczka := #indeks_mozliwych_ruchow;
END_FUNCTION

FUNCTION "sprawdz_ruch_gońca" : Int   // FC11, SCL
{ S7_Optimized_Access := 'TRUE' }
VERSION : 0.1
   VAR_INPUT
      szachownica : "Szachownica";
   END_VAR
   VAR_IN_OUT
      goniec : "Figura";
   END_VAR
   VAR_TEMP
      poz_temp : "Pozycja";
      indeks_mozliwych_ruchow : Int;
      wykonuj_petle : Bool;
   END_VAR
BEGIN
   #indeks_mozliwych_ruchow := 0;


   IF #goniec.kolor = 1 THEN
       #wykonuj_petle := TRUE;
       #poz_temp := #goniec.pozycja;
       WHILE #wykonuj_petle DO
           #poz_temp.x += 1;
           #poz_temp.y += 1;
           IF "sprawdz_czy_na_szachownicy"(#poz_temp) = true THEN
               IF "sprawdz_czy_wolne"(pozycja := #poz_temp, szachownica := #szachownica) = true THEN
                   IF "sprawdz_czy_ruch_możliwy"(figura:=#goniec, szachownica:=#szachownica, pozycja:=#poz_temp) = true  THEN
                       #goniec.mozliwe_ruchy[#indeks_mozliwych_ruchow] := #poz_temp;
                       #indeks_mozliwych_ruchow += 1;
                   END_IF;
               ELSIF "sprawdz_czy_zajete"(pozycja := #poz_temp, szachownica := #szachownica) = 1 THEN
                   IF "sprawdz_czy_ruch_możliwy"(figura:=#goniec, szachownica:=#szachownica, pozycja:=#poz_temp) = true  THEN
                       #goniec.mozliwe_ruchy[#indeks_mozliwych_ruchow] := #poz_temp;
                       #indeks_mozliwych_ruchow += 1;
                       #wykonuj_petle := false;
                   END_IF;
               ELSE
                   #wykonuj_petle := false;
               END_IF;
           ELSE
               #wykonuj_petle := false;
           END_IF;
       END_WHILE;
       #wykonuj_petle := TRUE;
       #poz_temp := #goniec.pozycja;
       WHILE #wykonuj_petle DO
           #poz_temp.x += 1;
           #poz_temp.y -= 1;
           IF "sprawdz_czy_na_szachownicy"(#poz_temp) = true THEN
               IF "sprawdz_czy_wolne"(pozycja := #poz_temp, szachownica := #szachownica) = true THEN
                   IF "sprawdz_czy_ruch_możliwy"(figura:=#goniec, szachownica:=#szachownica, pozycja:=#poz_temp) = true  THEN
                       #goniec.mozliwe_ruchy[#indeks_mozliwych_ruchow] := #poz_temp;
                       #indeks_mozliwych_ruchow += 1;
                   END_IF;
               ELSIF "sprawdz_czy_zajete"(pozycja := #poz_temp, szachownica := #szachownica) = 1 THEN
                   IF "sprawdz_czy_ruch_możliwy"(figura:=#goniec, szachownica:=#szachownica, pozycja:=#poz_temp) = true  THEN
                       #goniec.mozliwe_ruchy[#indeks_mozliwych_ruchow] := #poz_temp;
                       #indeks_mozliwych_ruchow += 1;
                       #wykonuj_petle:= false ;
                   END_IF;
               ELSE
                   #wykonuj_petle := false;
               END_IF;
           ELSE
               #wykonuj_petle := false;
           END_IF;
       END_WHILE;
       #wykonuj_petle := TRUE;
       #poz_temp := #goniec.pozycja;
       WHILE #wykonuj_petle DO
           #poz_temp.x -= 1;
           #poz_temp.y += 1;
           IF "sprawdz_czy_na_szachownicy"(#poz_temp) = true THEN
               IF "sprawdz_czy_wolne"(pozycja := #poz_temp, szachownica := #szachownica) = true THEN
                   IF "sprawdz_czy_ruch_możliwy"(figura:=#goniec, szachownica:=#szachownica, pozycja:=#poz_temp) = true  THEN
                       #goniec.mozliwe_ruchy[#indeks_mozliwych_ruchow] := #poz_temp;
                       #indeks_mozliwych_ruchow += 1;
                   END_IF;
               ELSIF "sprawdz_czy_zajete"(pozycja := #poz_temp, szachownica := #szachownica) = 1 THEN
                   IF "sprawdz_czy_ruch_możliwy"(figura:=#goniec, szachownica:=#szachownica, pozycja:=#poz_temp) = true  THEN
                       #goniec.mozliwe_ruchy[#indeks_mozliwych_ruchow] := #poz_temp;
                       #indeks_mozliwych_ruchow += 1;
                       #wykonuj_petle := false;
                   END_IF;
               ELSE
                   #wykonuj_petle := false;
               END_IF;
           ELSE
               #wykonuj_petle := false;
           END_IF;
       END_WHILE;
       #wykonuj_petle := TRUE;
       #poz_temp := #goniec.pozycja;
       WHILE #wykonuj_petle DO
           #poz_temp.x -= 1;
           #poz_temp.y -= 1;
           IF "sprawdz_czy_na_szachownicy"(#poz_temp) = true THEN
               IF "sprawdz_czy_wolne"(pozycja := #poz_temp, szachownica := #szachownica) = true THEN
                   IF "sprawdz_czy_ruch_możliwy"(figura:=#goniec, szachownica:=#szachownica, pozycja:=#poz_temp) = true  THEN
                       #goniec.mozliwe_ruchy[#indeks_mozliwych_ruchow] := #poz_temp;
                       #indeks_mozliwych_ruchow += 1;
                   END_IF;
               ELSIF "sprawdz_czy_zajete"(pozycja := #poz_temp, szachownica := #szachownica) = 1 THEN
                   IF "sprawdz_czy_ruch_możliwy"(figura:=#goniec, szachownica:=#szachownica, pozycja:=#poz_temp) = true  THEN
                       #goniec.mozliwe_ruchy[#indeks_mozliwych_ruchow] := #poz_temp;
                       #indeks_mozliwych_ruchow += 1;
                       #wykonuj_petle := false;
                   END_IF;
               ELSE
                   #wykonuj_petle := false;
               END_IF;
           ELSE
               #wykonuj_petle := false;
           END_IF;
       END_WHILE;


   ELSE
       #wykonuj_petle := TRUE;
       #poz_temp := #goniec.pozycja;
       WHILE #wykonuj_petle DO
           #poz_temp.x += 1;
           #poz_temp.y += 1;
           IF "sprawdz_czy_na_szachownicy"(#poz_temp) = true THEN
               IF "sprawdz_czy_wolne"(pozycja := #poz_temp, szachownica := #szachownica) = true THEN
                   IF "sprawdz_czy_ruch_możliwy"(figura:=#goniec, szachownica:=#szachownica, pozycja:=#poz_temp) = true  THEN
                       #goniec.mozliwe_ruchy[#indeks_mozliwych_ruchow] := #poz_temp;
                       #indeks_mozliwych_ruchow += 1;
                   END_IF;
               ELSIF "sprawdz_czy_zajete"(pozycja := #poz_temp, szachownica := #szachownica) = 2 THEN
                   IF "sprawdz_czy_ruch_możliwy"(figura:=#goniec, szachownica:=#szachownica, pozycja:=#poz_temp) = true  THEN
                       #goniec.mozliwe_ruchy[#indeks_mozliwych_ruchow] := #poz_temp;
                       #indeks_mozliwych_ruchow += 1;
                       #wykonuj_petle := false;
                   END_IF;
               ELSE
                   #wykonuj_petle := false;
               END_IF;
           ELSE
               #wykonuj_petle := false;
           END_IF;
       END_WHILE;
       #wykonuj_petle := TRUE;
       #poz_temp := #goniec.pozycja;
       WHILE #wykonuj_petle DO
           #poz_temp.x += 1;
           #poz_temp.y -= 1;
           IF "sprawdz_czy_na_szachownicy"(#poz_temp) = true THEN
               IF "sprawdz_czy_wolne"(pozycja := #poz_temp, szachownica := #szachownica) = true THEN
                   IF "sprawdz_czy_ruch_możliwy"(figura:=#goniec, szachownica:=#szachownica, pozycja:=#poz_temp) = true  THEN
                       #goniec.mozliwe_ruchy[#indeks_mozliwych_ruchow] := #poz_temp;
                       #indeks_mozliwych_ruchow += 1;
                   END_IF;
               ELSIF "sprawdz_czy_zajete"(pozycja := #poz_temp, szachownica := #szachownica) = 2 THEN
                   IF "sprawdz_czy_ruch_możliwy"(figura:=#goniec, szachownica:=#szachownica, pozycja:=#poz_temp) = true  THEN
                       #goniec.mozliwe_ruchy[#indeks_mozliwych_ruchow] := #poz_temp;
                       #indeks_mozliwych_ruchow += 1;
                       #wykonuj_petle := false;
                   END_IF;
               ELSE
                   #wykonuj_petle := false;
               END_IF;
           ELSE
               #wykonuj_petle := false;
           END_IF;
       END_WHILE;
       #wykonuj_petle := TRUE;
       #poz_temp := #goniec.pozycja;
       WHILE #wykonuj_petle DO
           #poz_temp.x -= 1;
           #poz_temp.y += 1;
           IF "sprawdz_czy_na_szachownicy"(#poz_temp) = true THEN
               IF "sprawdz_czy_wolne"(pozycja := #poz_temp, szachownica := #szachownica) = true THEN
                   IF "sprawdz_czy_ruch_możliwy"(figura:=#goniec, szachownica:=#szachownica, pozycja:=#poz_temp) = true  THEN
                       #goniec.mozliwe_ruchy[#indeks_mozliwych_ruchow] := #poz_temp;
                       #indeks_mozliwych_ruchow += 1;
                   END_IF;
               ELSIF "sprawdz_czy_zajete"(pozycja := #poz_temp, szachownica := #szachownica) = 2 THEN
                   IF "sprawdz_czy_ruch_możliwy"(figura:=#goniec, szachownica:=#szachownica, pozycja:=#poz_temp) = true  THEN
                       #goniec.mozliwe_ruchy[#indeks_mozliwych_ruchow] := #poz_temp;
                       #indeks_mozliwych_ruchow += 1;
                       #wykonuj_petle := false;
                   END_IF;
               ELSE
                   #wykonuj_petle := false;
               END_IF;
           ELSE
               #wykonuj_petle := false;
           END_IF;
       END_WHILE;
       #wykonuj_petle := TRUE;
       #poz_temp := #goniec.pozycja;
       WHILE #wykonuj_petle DO
           #poz_temp.x -= 1;
           #poz_temp.y -= 1;
           IF "sprawdz_czy_na_szachownicy"(#poz_temp) = true THEN
               IF "sprawdz_czy_wolne"(pozycja := #poz_temp, szachownica := #szachownica) = true THEN
                   IF "sprawdz_czy_ruch_możliwy"(figura:=#goniec, szachownica:=#szachownica, pozycja:=#poz_temp) = true  THEN
                       #goniec.mozliwe_ruchy[#indeks_mozliwych_ruchow] := #poz_temp;
                       #indeks_mozliwych_ruchow += 1;
                   END_IF;
               ELSIF "sprawdz_czy_zajete"(pozycja := #poz_temp, szachownica := #szachownica) = 2 THEN
                   IF "sprawdz_czy_ruch_możliwy"(figura:=#goniec, szachownica:=#szachownica, pozycja:=#poz_temp) = true  THEN
                       #goniec.mozliwe_ruchy[#indeks_mozliwych_ruchow] := #poz_temp;
                       #indeks_mozliwych_ruchow += 1;
                       #wykonuj_petle := false;
                   END_IF;
               ELSE
                   #wykonuj_petle := false;
               END_IF;
           ELSE
               #wykonuj_petle := false;
           END_IF;
       END_WHILE;
   END_IF;
   #sprawdz_ruch_gońca := #indeks_mozliwych_ruchow;
END_FUNCTION

FUNCTION "sprawdz_ruch_wieży" : Int   // FC12, SCL
{ S7_Optimized_Access := 'TRUE' }
VERSION : 0.1
   VAR_INPUT
      szachownica : "Szachownica";
   END_VAR
   VAR_IN_OUT
      wieza : "Figura";
   END_VAR
   VAR_TEMP
      poz_temp : "Pozycja";
      wykonuj_petle : Bool;
      indeks_mozliwych_ruchow : Int;
   END_VAR
BEGIN
   #indeks_mozliwych_ruchow := 0;


   IF #wieza.kolor = 1 THEN
       // ruch białych 
       // 
       //ruch poziomo i pionowo
       #wykonuj_petle := TRUE;
       #poz_temp := #wieza.pozycja;
       WHILE #wykonuj_petle DO
           #poz_temp.x += 1;
           #poz_temp.y += 0;
           IF "sprawdz_czy_na_szachownicy"(#poz_temp) = true THEN
               IF "sprawdz_czy_wolne"(pozycja := #poz_temp, szachownica := #szachownica) = true THEN
                   IF "sprawdz_czy_ruch_możliwy"(figura := #wieza, szachownica := #szachownica, pozycja := #poz_temp)  = true THEN
                       #wieza.mozliwe_ruchy[#indeks_mozliwych_ruchow] := #poz_temp;
                       #indeks_mozliwych_ruchow += 1;
                   END_IF;
               ELSIF "sprawdz_czy_zajete"(pozycja := #poz_temp, szachownica := #szachownica) = 1 THEN
                   IF "sprawdz_czy_ruch_możliwy"(figura := #wieza, szachownica := #szachownica, pozycja := #poz_temp)  = true THEN
                       #wieza.mozliwe_ruchy[#indeks_mozliwych_ruchow] := #poz_temp;
                       #indeks_mozliwych_ruchow += 1;
                       #wykonuj_petle := false;
                   END_IF;
               ELSE
                   #wykonuj_petle := false;
               END_IF;
           ELSE
               #wykonuj_petle := false;
           END_IF;
       END_WHILE;
       #wykonuj_petle := TRUE;
       #poz_temp := #wieza.pozycja;
       WHILE #wykonuj_petle DO
           #poz_temp.x += 0;
           #poz_temp.y += 1;
           IF "sprawdz_czy_na_szachownicy"(#poz_temp) = true THEN
               IF "sprawdz_czy_wolne"(pozycja := #poz_temp, szachownica := #szachownica) = true THEN
                   IF "sprawdz_czy_ruch_możliwy"(figura := #wieza, szachownica := #szachownica, pozycja := #poz_temp)  = true THEN
                       #wieza.mozliwe_ruchy[#indeks_mozliwych_ruchow] := #poz_temp;
                       #indeks_mozliwych_ruchow += 1;
                   END_IF;
               ELSIF "sprawdz_czy_zajete"(pozycja := #poz_temp, szachownica := #szachownica) = 1 THEN
                   IF "sprawdz_czy_ruch_możliwy"(figura := #wieza, szachownica := #szachownica, pozycja := #poz_temp) = true THEN
                       #wieza.mozliwe_ruchy[#indeks_mozliwych_ruchow] := #poz_temp;
                       #indeks_mozliwych_ruchow += 1;
                       #wykonuj_petle := false;
                   END_IF;
               ELSE
                   #wykonuj_petle := false;
               END_IF;
           ELSE
               #wykonuj_petle := false;
           END_IF;
       END_WHILE;
       #wykonuj_petle := TRUE;
       #poz_temp := #wieza.pozycja;
       WHILE #wykonuj_petle DO
           #poz_temp.x += -1;
           #poz_temp.y += 0;
           IF "sprawdz_czy_na_szachownicy"(#poz_temp) = true THEN
               IF "sprawdz_czy_wolne"(pozycja := #poz_temp, szachownica := #szachownica) = true THEN
                   IF "sprawdz_czy_ruch_możliwy"(figura := #wieza, szachownica := #szachownica, pozycja := #poz_temp)  = true THEN
                       #wieza.mozliwe_ruchy[#indeks_mozliwych_ruchow] := #poz_temp;
                       #indeks_mozliwych_ruchow += 1;
                   END_IF;
               ELSIF "sprawdz_czy_zajete"(pozycja := #poz_temp, szachownica := #szachownica) = 1 THEN
                   IF "sprawdz_czy_ruch_możliwy"(figura := #wieza, szachownica := #szachownica, pozycja := #poz_temp)  = true THEN
                       #wieza.mozliwe_ruchy[#indeks_mozliwych_ruchow] := #poz_temp;
                       #indeks_mozliwych_ruchow += 1;
                       #wykonuj_petle := false;
                   END_IF;
               ELSE
                   #wykonuj_petle := false;
               END_IF;
           ELSE
               #wykonuj_petle := false;
           END_IF;
       END_WHILE;
       #wykonuj_petle := TRUE;
       #poz_temp := #wieza.pozycja;
       WHILE #wykonuj_petle DO
           #poz_temp.x += 0;
           #poz_temp.y += -1;
           IF "sprawdz_czy_na_szachownicy"(#poz_temp) = true THEN
               IF "sprawdz_czy_wolne"(pozycja := #poz_temp, szachownica := #szachownica) = true THEN
                   IF "sprawdz_czy_ruch_możliwy"(figura := #wieza, szachownica := #szachownica, pozycja := #poz_temp)  = true THEN
                       #wieza.mozliwe_ruchy[#indeks_mozliwych_ruchow] := #poz_temp;
                       #indeks_mozliwych_ruchow += 1;
                   END_IF;
               ELSIF "sprawdz_czy_zajete"(pozycja := #poz_temp, szachownica := #szachownica) = 1 THEN
                   IF "sprawdz_czy_ruch_możliwy"(figura := #wieza, szachownica := #szachownica, pozycja := #poz_temp)  = true THEN
                       #wieza.mozliwe_ruchy[#indeks_mozliwych_ruchow] := #poz_temp;
                       #indeks_mozliwych_ruchow += 1;
                       #wykonuj_petle := false;
                   END_IF;
               ELSE
                   #wykonuj_petle := false;
               END_IF;
           ELSE
               #wykonuj_petle := false;
           END_IF;
       END_WHILE;


   ELSE
       //ruch czarnych
       //
       //ruch poziomo i pionowo
       #wykonuj_petle := TRUE;
       #poz_temp := #wieza.pozycja;
       WHILE #wykonuj_petle DO
           #poz_temp.x += 1;
           #poz_temp.y += 0;
           IF "sprawdz_czy_na_szachownicy"(#poz_temp) = true THEN
               IF "sprawdz_czy_wolne"(pozycja := #poz_temp, szachownica := #szachownica) = true THEN
                   IF "sprawdz_czy_ruch_możliwy"(figura := #wieza, szachownica := #szachownica, pozycja := #poz_temp)  = true THEN
                       #wieza.mozliwe_ruchy[#indeks_mozliwych_ruchow] := #poz_temp;
                       #indeks_mozliwych_ruchow += 1;
                   END_IF;
               ELSIF "sprawdz_czy_zajete"(pozycja := #poz_temp, szachownica := #szachownica) = 2 THEN
                   IF "sprawdz_czy_ruch_możliwy"(figura := #wieza, szachownica := #szachownica, pozycja := #poz_temp)  = true THEN
                       #wieza.mozliwe_ruchy[#indeks_mozliwych_ruchow] := #poz_temp;
                       #indeks_mozliwych_ruchow += 1;
                       #wykonuj_petle := false;
                   END_IF;
               ELSE
                   #wykonuj_petle := false;
               END_IF;
           ELSE
               #wykonuj_petle := false;
           END_IF;
       END_WHILE;
       #wykonuj_petle := TRUE;
       #poz_temp := #wieza.pozycja;
       WHILE #wykonuj_petle DO
           #poz_temp.x += 0;
           #poz_temp.y += 1;
           IF "sprawdz_czy_na_szachownicy"(#poz_temp) = true THEN
               IF "sprawdz_czy_wolne"(pozycja := #poz_temp, szachownica := #szachownica) = true THEN
                   IF "sprawdz_czy_ruch_możliwy"(figura := #wieza, szachownica := #szachownica, pozycja := #poz_temp)  = true THEN
                       #wieza.mozliwe_ruchy[#indeks_mozliwych_ruchow] := #poz_temp;
                       #indeks_mozliwych_ruchow += 1;
                   END_IF;
               ELSIF "sprawdz_czy_zajete"(pozycja := #poz_temp, szachownica := #szachownica) = 2 THEN
                   IF "sprawdz_czy_ruch_możliwy"(figura := #wieza, szachownica := #szachownica, pozycja := #poz_temp)  = true THEN
                       #wieza.mozliwe_ruchy[#indeks_mozliwych_ruchow] := #poz_temp;
                       #indeks_mozliwych_ruchow += 1;
                       #wykonuj_petle := false;
                   END_IF;
               ELSE
                   #wykonuj_petle := false;
               END_IF;
           ELSE
               #wykonuj_petle := false;
           END_IF;
       END_WHILE;
       #wykonuj_petle := TRUE;
       #poz_temp := #wieza.pozycja;
       WHILE #wykonuj_petle DO
           #poz_temp.x += -1;
           #poz_temp.y += 0;
           IF "sprawdz_czy_na_szachownicy"(#poz_temp) = true THEN
               IF "sprawdz_czy_wolne"(pozycja := #poz_temp, szachownica := #szachownica) = true THEN
                   IF "sprawdz_czy_ruch_możliwy"(figura := #wieza, szachownica := #szachownica, pozycja := #poz_temp)  = true THEN
                       #wieza.mozliwe_ruchy[#indeks_mozliwych_ruchow] := #poz_temp;
                       #indeks_mozliwych_ruchow += 1;
                   END_IF;
               ELSIF "sprawdz_czy_zajete"(pozycja := #poz_temp, szachownica := #szachownica) = 2 THEN
                   IF "sprawdz_czy_ruch_możliwy"(figura := #wieza, szachownica := #szachownica, pozycja := #poz_temp)  = true THEN
                       #wieza.mozliwe_ruchy[#indeks_mozliwych_ruchow] := #poz_temp;
                       #indeks_mozliwych_ruchow += 1;
                       #wykonuj_petle := false;
                   END_IF;
               ELSE
                   #wykonuj_petle := false;
               END_IF;
           ELSE
               #wykonuj_petle := false;
           END_IF;
       END_WHILE;
       #wykonuj_petle := TRUE;
       #poz_temp := #wieza.pozycja;
       WHILE #wykonuj_petle DO
           #poz_temp.x += 0;
           #poz_temp.y += -1;
           IF "sprawdz_czy_na_szachownicy"(#poz_temp) = true THEN
               IF "sprawdz_czy_wolne"(pozycja := #poz_temp, szachownica := #szachownica) = true THEN
                   IF "sprawdz_czy_ruch_możliwy"(figura := #wieza, szachownica := #szachownica, pozycja := #poz_temp)  = true THEN
                       #wieza.mozliwe_ruchy[#indeks_mozliwych_ruchow] := #poz_temp;
                       #indeks_mozliwych_ruchow += 1;
                   END_IF;
               ELSIF "sprawdz_czy_zajete"(pozycja := #poz_temp, szachownica := #szachownica) = 2 THEN
                   IF "sprawdz_czy_ruch_możliwy"(figura := #wieza, szachownica := #szachownica, pozycja := #poz_temp)  = true THEN
                       #wieza.mozliwe_ruchy[#indeks_mozliwych_ruchow] := #poz_temp;
                       #indeks_mozliwych_ruchow += 1;
                       #wykonuj_petle := false;
                   END_IF;
               ELSE
                   #wykonuj_petle := false;
               END_IF;
           ELSE
               #wykonuj_petle := false;
           END_IF;
       END_WHILE;
   END_IF;
   #sprawdz_ruch_wieży := #indeks_mozliwych_ruchow;
END_FUNCTION

FUNCTION "sprawdz_ruch_króla" : Int   // FC13, SCL
{ S7_Optimized_Access := 'TRUE' }
VERSION : 0.1
   VAR_INPUT
      szachownica : "Szachownica";
   END_VAR
   VAR_IN_OUT
      krol : "Figura";
   END_VAR
   VAR_TEMP
      poz_temp : "Pozycja";
      indeks_mozliwych_ruchow : Int;
   END_VAR
BEGIN
   #indeks_mozliwych_ruchow := 0;
   IF #krol.kolor = 1 THEN
       // ruchy króla bialego we wszystkich kierunkach
       #poz_temp := #krol.pozycja;
       #poz_temp.x := #krol.pozycja.x;
       #poz_temp.y := #krol.pozycja.y + 1;
       IF "sprawdz_czy_na_szachownicy"(#poz_temp) = true THEN
           IF "sprawdz_czy_wolne"(pozycja := #poz_temp, szachownica := #szachownica) = true THEN
               IF "sprawdz_czy_ruch_możliwy"(figura := #krol, szachownica := #szachownica, pozycja := #poz_temp) = true  THEN
                   #krol.mozliwe_ruchy[#indeks_mozliwych_ruchow] := #poz_temp;
                   #indeks_mozliwych_ruchow += 1;
               END_IF;
           ELSIF "sprawdz_czy_zajete"(pozycja := #poz_temp, szachownica := #szachownica) = 1 THEN
               IF "sprawdz_czy_ruch_możliwy"(figura := #krol, szachownica := #szachownica, pozycja := #poz_temp) = true  THEN
                   #krol.mozliwe_ruchy[#indeks_mozliwych_ruchow] := #poz_temp;
                   #indeks_mozliwych_ruchow += 1;
               END_IF;
           END_IF;
       END_IF;
       #poz_temp := #krol.pozycja;
       #poz_temp.x := #krol.pozycja.x + 1;
       #poz_temp.y := #krol.pozycja.y + 1;
       IF "sprawdz_czy_na_szachownicy"(#poz_temp) = true THEN
           IF "sprawdz_czy_wolne"(pozycja := #poz_temp, szachownica := #szachownica) = true THEN
               IF "sprawdz_czy_ruch_możliwy"(figura := #krol, szachownica := #szachownica, pozycja := #poz_temp) = true  THEN
                   #krol.mozliwe_ruchy[#indeks_mozliwych_ruchow] := #poz_temp;
                   #indeks_mozliwych_ruchow += 1;
               END_IF;
           ELSIF "sprawdz_czy_zajete"(pozycja := #poz_temp, szachownica := #szachownica) = 1 THEN
               IF "sprawdz_czy_ruch_możliwy"(figura := #krol, szachownica := #szachownica, pozycja := #poz_temp) = true  THEN
                   #krol.mozliwe_ruchy[#indeks_mozliwych_ruchow] := #poz_temp;
                   #indeks_mozliwych_ruchow += 1;
               END_IF;
           END_IF;
       END_IF;
       #poz_temp := #krol.pozycja;
       #poz_temp.x := #krol.pozycja.x + 1;
       #poz_temp.y := #krol.pozycja.y;
       IF "sprawdz_czy_na_szachownicy"(#poz_temp) = true THEN
           IF "sprawdz_czy_wolne"(pozycja := #poz_temp, szachownica := #szachownica) = true THEN
               IF "sprawdz_czy_ruch_możliwy"(figura := #krol, szachownica := #szachownica, pozycja := #poz_temp) = true  THEN
                   #krol.mozliwe_ruchy[#indeks_mozliwych_ruchow] := #poz_temp;
                   #indeks_mozliwych_ruchow += 1;
               END_IF;
           ELSIF "sprawdz_czy_zajete"(pozycja := #poz_temp, szachownica := #szachownica) = 1 THEN
               IF "sprawdz_czy_ruch_możliwy"(figura := #krol, szachownica := #szachownica, pozycja := #poz_temp) = true  THEN
                   #krol.mozliwe_ruchy[#indeks_mozliwych_ruchow] := #poz_temp;
                   #indeks_mozliwych_ruchow += 1;
               END_IF;
           END_IF;
       END_IF;
       #poz_temp := #krol.pozycja;
       #poz_temp.x := #krol.pozycja.x + 1;
       #poz_temp.y := #krol.pozycja.y - 1;
       IF "sprawdz_czy_na_szachownicy"(#poz_temp) = true THEN
           IF "sprawdz_czy_wolne"(pozycja := #poz_temp, szachownica := #szachownica) = true THEN
               IF "sprawdz_czy_ruch_możliwy"(figura := #krol, szachownica := #szachownica, pozycja := #poz_temp) = true  THEN
                   #krol.mozliwe_ruchy[#indeks_mozliwych_ruchow] := #poz_temp;
                   #indeks_mozliwych_ruchow += 1;
               END_IF;
           ELSIF "sprawdz_czy_zajete"(pozycja := #poz_temp, szachownica := #szachownica) = 1 THEN
               IF "sprawdz_czy_ruch_możliwy"(figura := #krol, szachownica := #szachownica, pozycja := #poz_temp) = true  THEN
                   #krol.mozliwe_ruchy[#indeks_mozliwych_ruchow] := #poz_temp;
                   #indeks_mozliwych_ruchow += 1;
               END_IF;
           END_IF;
       END_IF;
       #poz_temp := #krol.pozycja;
       #poz_temp.x := #krol.pozycja.x;
       #poz_temp.y := #krol.pozycja.y - 1;
       IF "sprawdz_czy_na_szachownicy"(#poz_temp) = true THEN
           IF "sprawdz_czy_wolne"(pozycja := #poz_temp, szachownica := #szachownica) = true THEN
               IF "sprawdz_czy_ruch_możliwy"(figura := #krol, szachownica := #szachownica, pozycja := #poz_temp) = true  THEN
                   #krol.mozliwe_ruchy[#indeks_mozliwych_ruchow] := #poz_temp;
                   #indeks_mozliwych_ruchow += 1;
               END_IF;
           ELSIF "sprawdz_czy_zajete"(pozycja := #poz_temp, szachownica := #szachownica) = 1 THEN
               IF "sprawdz_czy_ruch_możliwy"(figura := #krol, szachownica := #szachownica, pozycja := #poz_temp) = true  THEN
                   #krol.mozliwe_ruchy[#indeks_mozliwych_ruchow] := #poz_temp;
                   #indeks_mozliwych_ruchow += 1;
               END_IF;
           END_IF;
       END_IF;
       #poz_temp := #krol.pozycja;
       #poz_temp.x := #krol.pozycja.x - 1;
       #poz_temp.y := #krol.pozycja.y - 1;
       IF "sprawdz_czy_na_szachownicy"(#poz_temp) = true THEN
           IF "sprawdz_czy_wolne"(pozycja := #poz_temp, szachownica := #szachownica) = true THEN
               IF "sprawdz_czy_ruch_możliwy"(figura := #krol, szachownica := #szachownica, pozycja := #poz_temp) = true  THEN
                   #krol.mozliwe_ruchy[#indeks_mozliwych_ruchow] := #poz_temp;
                   #indeks_mozliwych_ruchow += 1;
               END_IF;
           ELSIF "sprawdz_czy_zajete"(pozycja := #poz_temp, szachownica := #szachownica) = 1 THEN
               IF "sprawdz_czy_ruch_możliwy"(figura := #krol, szachownica := #szachownica, pozycja := #poz_temp) = true  THEN
                   #krol.mozliwe_ruchy[#indeks_mozliwych_ruchow] := #poz_temp;
                   #indeks_mozliwych_ruchow += 1;
               END_IF;
           END_IF;
       END_IF;
       #poz_temp := #krol.pozycja;
       #poz_temp.x := #krol.pozycja.x - 1;
       #poz_temp.y := #krol.pozycja.y;
       IF "sprawdz_czy_na_szachownicy"(#poz_temp) = true THEN
           IF "sprawdz_czy_wolne"(pozycja := #poz_temp, szachownica := #szachownica) = true THEN
               IF "sprawdz_czy_ruch_możliwy"(figura := #krol, szachownica := #szachownica, pozycja := #poz_temp) = true  THEN
                   #krol.mozliwe_ruchy[#indeks_mozliwych_ruchow] := #poz_temp;
                   #indeks_mozliwych_ruchow += 1;
               END_IF;
           ELSIF "sprawdz_czy_zajete"(pozycja := #poz_temp, szachownica := #szachownica) = 1 THEN
               IF "sprawdz_czy_ruch_możliwy"(figura := #krol, szachownica := #szachownica, pozycja := #poz_temp) = true  THEN
                   #krol.mozliwe_ruchy[#indeks_mozliwych_ruchow] := #poz_temp;
                   #indeks_mozliwych_ruchow += 1;
               END_IF;
           END_IF;
       END_IF;
       #poz_temp := #krol.pozycja;
       #poz_temp.x := #krol.pozycja.x - 1;
       #poz_temp.y := #krol.pozycja.y + 1;
       IF "sprawdz_czy_na_szachownicy"(#poz_temp) = true THEN
           IF "sprawdz_czy_wolne"(pozycja := #poz_temp, szachownica := #szachownica) = true THEN
               IF "sprawdz_czy_ruch_możliwy"(figura := #krol, szachownica := #szachownica, pozycja := #poz_temp) = true  THEN
                   #krol.mozliwe_ruchy[#indeks_mozliwych_ruchow] := #poz_temp;
                   #indeks_mozliwych_ruchow += 1;
               END_IF;
           ELSIF "sprawdz_czy_zajete"(pozycja := #poz_temp, szachownica := #szachownica) = 1 THEN
               IF "sprawdz_czy_ruch_możliwy"(figura := #krol, szachownica := #szachownica, pozycja := #poz_temp) = true  THEN
                   #krol.mozliwe_ruchy[#indeks_mozliwych_ruchow] := #poz_temp;
                   #indeks_mozliwych_ruchow += 1;
               END_IF;
           END_IF;
       END_IF;
       // roszada
       IF NOT "Status_rozgrywki".szach_biale THEN
           IF #krol.poczatkowa_pozycja AND #szachownica.figury[0].poczatkowa_pozycja THEN
               #poz_temp := #krol.pozycja;
               #poz_temp.x := #poz_temp.x - 1;
               IF "sprawdz_czy_wolne"(szachownica := #szachownica, pozycja := #poz_temp) AND
                   "sprawdz_czy_ruch_możliwy"(figura := #krol, szachownica := #szachownica, pozycja := #poz_temp) = true THEN
                   #poz_temp.x := #poz_temp.x - 1;
                   IF "sprawdz_czy_wolne"(szachownica := #szachownica, pozycja := #poz_temp) AND
                       "sprawdz_czy_ruch_możliwy"(figura := #krol, szachownica := #szachownica, pozycja := #poz_temp) = true THEN
                       #poz_temp.x := #poz_temp.x - 1;
                       IF "sprawdz_czy_wolne"(szachownica := #szachownica, pozycja := #poz_temp) THEN
                           #poz_temp.x := #poz_temp.x + 1;
                           #krol.mozliwe_ruchy[#indeks_mozliwych_ruchow] := #poz_temp;
                           #indeks_mozliwych_ruchow += 1;

                       END_IF;
                   END_IF;
               END_IF;
           END_IF;
           IF #krol.poczatkowa_pozycja AND #szachownica.figury[7].poczatkowa_pozycja THEN
               #poz_temp := #krol.pozycja;
               #poz_temp.x := #poz_temp.x + 1;
               IF "sprawdz_czy_wolne"(szachownica := #szachownica, pozycja := #poz_temp) AND
                   "sprawdz_czy_ruch_możliwy"(figura := #krol, szachownica := #szachownica, pozycja := #poz_temp) = true THEN
                   #poz_temp.x := #poz_temp.x + 1;
                   IF "sprawdz_czy_wolne"(szachownica := #szachownica, pozycja := #poz_temp) AND
                       "sprawdz_czy_ruch_możliwy"(figura := #krol, szachownica := #szachownica, pozycja := #poz_temp) = true THEN
                       #krol.mozliwe_ruchy[#indeks_mozliwych_ruchow] := #poz_temp;
                       #indeks_mozliwych_ruchow += 1;
                   END_IF;
               END_IF;
           END_IF;
       END_IF;



   ELSE
       // ruchy króla bialego we wszystkich kierunkach
       #poz_temp := #krol.pozycja;
       #poz_temp.x := #krol.pozycja.x;
       #poz_temp.y := #krol.pozycja.y + 1;
       IF "sprawdz_czy_na_szachownicy"(#poz_temp) = true THEN
           IF "sprawdz_czy_wolne"(pozycja := #poz_temp, szachownica := #szachownica) = true THEN
               IF "sprawdz_czy_ruch_możliwy"(figura := #krol, szachownica := #szachownica, pozycja := #poz_temp) = true  THEN
                   #poz_temp.x := #poz_temp.x + 1;
                   #krol.mozliwe_ruchy[#indeks_mozliwych_ruchow] := #poz_temp;
                   #indeks_mozliwych_ruchow += 1;
               END_IF;
           ELSIF "sprawdz_czy_zajete"(pozycja := #poz_temp, szachownica := #szachownica) = 2 THEN
               IF "sprawdz_czy_ruch_możliwy"(figura := #krol, szachownica := #szachownica, pozycja := #poz_temp) = true  THEN
                   #krol.mozliwe_ruchy[#indeks_mozliwych_ruchow] := #poz_temp;
                   #indeks_mozliwych_ruchow += 1;
               END_IF;
           END_IF;
       END_IF;
       #poz_temp := #krol.pozycja;
       #poz_temp.x := #krol.pozycja.x + 1;
       #poz_temp.y := #krol.pozycja.y + 1;
       IF "sprawdz_czy_na_szachownicy"(#poz_temp) = true THEN
           IF "sprawdz_czy_wolne"(pozycja := #poz_temp, szachownica := #szachownica) = true THEN
               IF "sprawdz_czy_ruch_możliwy"(figura := #krol, szachownica := #szachownica, pozycja := #poz_temp) = true  THEN
                   #krol.mozliwe_ruchy[#indeks_mozliwych_ruchow] := #poz_temp;
                   #indeks_mozliwych_ruchow += 1;
               END_IF;
           ELSIF "sprawdz_czy_zajete"(pozycja := #poz_temp, szachownica := #szachownica) = 2 THEN
               IF "sprawdz_czy_ruch_możliwy"(figura := #krol, szachownica := #szachownica, pozycja := #poz_temp) = true  THEN
                   #krol.mozliwe_ruchy[#indeks_mozliwych_ruchow] := #poz_temp;
                   #indeks_mozliwych_ruchow += 1;
               END_IF;
           END_IF;
       END_IF;
       #poz_temp := #krol.pozycja;
       #poz_temp.x := #krol.pozycja.x + 1;
       #poz_temp.y := #krol.pozycja.y;
       IF "sprawdz_czy_na_szachownicy"(#poz_temp) = true THEN
           IF "sprawdz_czy_wolne"(pozycja := #poz_temp, szachownica := #szachownica) = true THEN
               IF "sprawdz_czy_ruch_możliwy"(figura := #krol, szachownica := #szachownica, pozycja := #poz_temp) = true  THEN
                   #krol.mozliwe_ruchy[#indeks_mozliwych_ruchow] := #poz_temp;
                   #indeks_mozliwych_ruchow += 1;
               END_IF;
           ELSIF "sprawdz_czy_zajete"(pozycja := #poz_temp, szachownica := #szachownica) = 2 THEN
               IF "sprawdz_czy_ruch_możliwy"(figura := #krol, szachownica := #szachownica, pozycja := #poz_temp) = true  THEN
                   #krol.mozliwe_ruchy[#indeks_mozliwych_ruchow] := #poz_temp;
                   #indeks_mozliwych_ruchow += 1;
               END_IF;
           END_IF;
       END_IF;
       #poz_temp := #krol.pozycja;
       #poz_temp.x := #krol.pozycja.x + 1;
       #poz_temp.y := #krol.pozycja.y - 1;
       IF "sprawdz_czy_na_szachownicy"(#poz_temp) = true THEN
           IF "sprawdz_czy_wolne"(pozycja := #poz_temp, szachownica := #szachownica) = true THEN
               IF "sprawdz_czy_ruch_możliwy"(figura := #krol, szachownica := #szachownica, pozycja := #poz_temp) = true  THEN
                   #krol.mozliwe_ruchy[#indeks_mozliwych_ruchow] := #poz_temp;
                   #indeks_mozliwych_ruchow += 1;
               END_IF;
           ELSIF "sprawdz_czy_zajete"(pozycja := #poz_temp, szachownica := #szachownica) = 2 THEN
               IF "sprawdz_czy_ruch_możliwy"(figura := #krol, szachownica := #szachownica, pozycja := #poz_temp) = true  THEN
                   #krol.mozliwe_ruchy[#indeks_mozliwych_ruchow] := #poz_temp;
                   #indeks_mozliwych_ruchow += 1;
               END_IF;
           END_IF;
       END_IF;
       #poz_temp := #krol.pozycja;
       #poz_temp.x := #krol.pozycja.x;
       #poz_temp.y := #krol.pozycja.y - 1;
       IF "sprawdz_czy_na_szachownicy"(#poz_temp) = true THEN
           IF "sprawdz_czy_wolne"(pozycja := #poz_temp, szachownica := #szachownica) = true THEN
               IF "sprawdz_czy_ruch_możliwy"(figura := #krol, szachownica := #szachownica, pozycja := #poz_temp) = true  THEN
                   #krol.mozliwe_ruchy[#indeks_mozliwych_ruchow] := #poz_temp;
                   #indeks_mozliwych_ruchow += 1;
               END_IF;
           ELSIF "sprawdz_czy_zajete"(pozycja := #poz_temp, szachownica := #szachownica) = 2 THEN
               IF "sprawdz_czy_ruch_możliwy"(figura := #krol, szachownica := #szachownica, pozycja := #poz_temp) = true  THEN
                   #krol.mozliwe_ruchy[#indeks_mozliwych_ruchow] := #poz_temp;
                   #indeks_mozliwych_ruchow += 1;
               END_IF;
           END_IF;
       END_IF;
       #poz_temp := #krol.pozycja;
       #poz_temp.x := #krol.pozycja.x - 1;
       #poz_temp.y := #krol.pozycja.y - 1;
       IF "sprawdz_czy_na_szachownicy"(#poz_temp) = true THEN
           IF "sprawdz_czy_wolne"(pozycja := #poz_temp, szachownica := #szachownica) = true THEN
               IF "sprawdz_czy_ruch_możliwy"(figura := #krol, szachownica := #szachownica, pozycja := #poz_temp) = true  THEN
                   #krol.mozliwe_ruchy[#indeks_mozliwych_ruchow] := #poz_temp;
                   #indeks_mozliwych_ruchow += 1;
               END_IF;
           ELSIF "sprawdz_czy_zajete"(pozycja := #poz_temp, szachownica := #szachownica) = 2 THEN
               IF "sprawdz_czy_ruch_możliwy"(figura := #krol, szachownica := #szachownica, pozycja := #poz_temp) = true  THEN
                   #krol.mozliwe_ruchy[#indeks_mozliwych_ruchow] := #poz_temp;
                   #indeks_mozliwych_ruchow += 1;
               END_IF;
           END_IF;
       END_IF;
       #poz_temp := #krol.pozycja;
       #poz_temp.x := #krol.pozycja.x - 1;
       #poz_temp.y := #krol.pozycja.y;
       IF "sprawdz_czy_na_szachownicy"(#poz_temp) = true THEN
           IF "sprawdz_czy_wolne"(pozycja := #poz_temp, szachownica := #szachownica) = true THEN
               IF "sprawdz_czy_ruch_możliwy"(figura := #krol, szachownica := #szachownica, pozycja := #poz_temp) = true  THEN
                   #krol.mozliwe_ruchy[#indeks_mozliwych_ruchow] := #poz_temp;
                   #indeks_mozliwych_ruchow += 1;
               END_IF;
           ELSIF "sprawdz_czy_zajete"(pozycja := #poz_temp, szachownica := #szachownica) = 2 THEN
               IF "sprawdz_czy_ruch_możliwy"(figura := #krol, szachownica := #szachownica, pozycja := #poz_temp) = true  THEN
                   #krol.mozliwe_ruchy[#indeks_mozliwych_ruchow] := #poz_temp;
                   #indeks_mozliwych_ruchow += 1;
               END_IF;
           END_IF;
       END_IF;
       #poz_temp := #krol.pozycja;
       #poz_temp.x := #krol.pozycja.x - 1;
       #poz_temp.y := #krol.pozycja.y + 1;
       IF "sprawdz_czy_na_szachownicy"(#poz_temp) = true THEN
           IF "sprawdz_czy_wolne"(pozycja := #poz_temp, szachownica := #szachownica) = true THEN
               IF "sprawdz_czy_ruch_możliwy"(figura := #krol, szachownica := #szachownica, pozycja := #poz_temp) = true  THEN
                   #krol.mozliwe_ruchy[#indeks_mozliwych_ruchow] := #poz_temp;
                   #indeks_mozliwych_ruchow += 1;
               END_IF;
           ELSIF "sprawdz_czy_zajete"(pozycja := #poz_temp, szachownica := #szachownica) = 2 THEN
               IF "sprawdz_czy_ruch_możliwy"(figura := #krol, szachownica := #szachownica, pozycja := #poz_temp) = true  THEN
                   #krol.mozliwe_ruchy[#indeks_mozliwych_ruchow] := #poz_temp;
                   #indeks_mozliwych_ruchow += 1;
               END_IF;
           END_IF;
       END_IF;

       // roszada
       IF NOT "Status_rozgrywki".szach_czarne THEN
           IF #krol.poczatkowa_pozycja AND #szachownica.figury[24].poczatkowa_pozycja THEN
               #poz_temp := #krol.pozycja;
               #poz_temp.x :=#poz_temp.x - 1;
               IF "sprawdz_czy_wolne"(szachownica := #szachownica, pozycja := #poz_temp) AND
                   "sprawdz_czy_ruch_możliwy"(figura := #krol, szachownica := #szachownica, pozycja := #poz_temp) = true THEN
                   #poz_temp.x :=#poz_temp.x- 1;
                   IF "sprawdz_czy_wolne"(szachownica := #szachownica, pozycja := #poz_temp) AND
                       "sprawdz_czy_ruch_możliwy"(figura := #krol, szachownica := #szachownica, pozycja := #poz_temp) = true THEN
                       #poz_temp.x :=#poz_temp.x - 1;
                       IF "sprawdz_czy_wolne"(szachownica := #szachownica, pozycja := #poz_temp) THEN
                           #poz_temp.x := #poz_temp.x +1 ;
                           #krol.mozliwe_ruchy[#indeks_mozliwych_ruchow] := #poz_temp;
                           #indeks_mozliwych_ruchow += 1;

                       END_IF;
                   END_IF;
               END_IF;
           END_IF;
           IF #krol.poczatkowa_pozycja AND #szachownica.figury[31].poczatkowa_pozycja THEN
               #poz_temp := #krol.pozycja;
               #poz_temp.x :=#poz_temp.x + 1;
               IF "sprawdz_czy_wolne"(szachownica := #szachownica, pozycja := #poz_temp) AND
                   "sprawdz_czy_ruch_możliwy"(figura := #krol, szachownica := #szachownica, pozycja := #poz_temp) = true THEN
                   #poz_temp.x :=#poz_temp.x + 1;
                   IF "sprawdz_czy_wolne"(szachownica := #szachownica, pozycja := #poz_temp) AND
                       "sprawdz_czy_ruch_możliwy"(figura := #krol, szachownica := #szachownica, pozycja := #poz_temp) = true THEN
                        #krol.mozliwe_ruchy[#indeks_mozliwych_ruchow] := #poz_temp;
                        #indeks_mozliwych_ruchow += 1;
                   END_IF;
               END_IF;
           END_IF;
       END_IF;
   END_IF;


   #sprawdz_ruch_króla := #indeks_mozliwych_ruchow;
END_FUNCTION

FUNCTION "sprawdz_ruch_hetmana" : Int   // FC14, SCL
{ S7_Optimized_Access := 'TRUE' }
VERSION : 0.1
   VAR_INPUT
      szachownica : "Szachownica";
   END_VAR
   VAR_IN_OUT
      hetman : "Figura";
   END_VAR
   VAR_TEMP
      poz_temp : "Pozycja";
      wykonuj_petle : Bool;
      indeks_mozliwych_ruchow : Int;
   END_VAR
BEGIN
   #indeks_mozliwych_ruchow := 0;

   #poz_temp := #hetman.pozycja;
   IF #hetman.kolor = 1 THEN
       // ruch białych 
       // 
       //ruch po skosie 
       #wykonuj_petle := TRUE;
       #poz_temp := #hetman.pozycja;
       WHILE #wykonuj_petle DO
           #poz_temp.x += 1;
           #poz_temp.y += 1;
           IF "sprawdz_czy_na_szachownicy"(#poz_temp) = true THEN
               IF "sprawdz_czy_wolne"(pozycja := #poz_temp, szachownica := #szachownica) = true THEN
                       IF "sprawdz_czy_ruch_możliwy"(figura := #hetman, szachownica := #szachownica, pozycja := #poz_temp) = true  THEN
                       #hetman.mozliwe_ruchy[#indeks_mozliwych_ruchow] := #poz_temp;
                       #indeks_mozliwych_ruchow += 1;
                       END_IF;
                   ELSIF "sprawdz_czy_zajete"(pozycja := #poz_temp, szachownica := #szachownica) = 1 THEN
                       IF "sprawdz_czy_ruch_możliwy"(figura := #hetman, szachownica := #szachownica, pozycja := #poz_temp) = true  THEN
                           #hetman.mozliwe_ruchy[#indeks_mozliwych_ruchow] := #poz_temp;
                           #indeks_mozliwych_ruchow += 1;
                           #wykonuj_petle := false;
                       END_IF;
                   ELSE
                       #wykonuj_petle := false;
                END_IF;
           ELSE
               #wykonuj_petle := false;
           END_IF;
       END_WHILE;
       #wykonuj_petle := TRUE;
       #poz_temp := #hetman.pozycja;
       WHILE #wykonuj_petle DO
           #poz_temp.x += 1;
           #poz_temp.y -= 1;
           IF "sprawdz_czy_na_szachownicy"(#poz_temp) = true THEN
               IF "sprawdz_czy_wolne"(pozycja := #poz_temp, szachownica := #szachownica) = true THEN
                   IF "sprawdz_czy_ruch_możliwy"(figura := #hetman, szachownica := #szachownica, pozycja := #poz_temp) = true  THEN
                       #hetman.mozliwe_ruchy[#indeks_mozliwych_ruchow] := #poz_temp;
                       #indeks_mozliwych_ruchow += 1;
                   END_IF; 
               ELSIF "sprawdz_czy_zajete"(pozycja := #poz_temp, szachownica := #szachownica) = 1 THEN
                   IF "sprawdz_czy_ruch_możliwy"(figura := #hetman, szachownica := #szachownica, pozycja := #poz_temp) = true  THEN
                       #hetman.mozliwe_ruchy[#indeks_mozliwych_ruchow] := #poz_temp;
                       #indeks_mozliwych_ruchow += 1;
                       #wykonuj_petle := false;
                   END_IF;
               ELSE
                   #wykonuj_petle := false;
               END_IF;
           ELSE
               #wykonuj_petle := false;
           END_IF;
       END_WHILE;
       #wykonuj_petle := TRUE;
       #poz_temp := #hetman.pozycja;
       WHILE #wykonuj_petle DO
           #poz_temp.x -= 1;
           #poz_temp.y += 1;
           IF "sprawdz_czy_na_szachownicy"(#poz_temp) = true THEN
               IF "sprawdz_czy_wolne"(pozycja := #poz_temp, szachownica := #szachownica) = true THEN
                   IF "sprawdz_czy_ruch_możliwy"(figura := #hetman, szachownica := #szachownica, pozycja := #poz_temp) = true  THEN
                       #hetman.mozliwe_ruchy[#indeks_mozliwych_ruchow] := #poz_temp;
                       #indeks_mozliwych_ruchow += 1;
                   END_IF;
               ELSIF "sprawdz_czy_zajete"(pozycja := #poz_temp, szachownica := #szachownica) = 1 THEN
                   IF "sprawdz_czy_ruch_możliwy"(figura := #hetman, szachownica := #szachownica, pozycja := #poz_temp) = true  THEN
                       #hetman.mozliwe_ruchy[#indeks_mozliwych_ruchow] := #poz_temp;
                       #indeks_mozliwych_ruchow += 1;
                       #wykonuj_petle := false;
                   END_IF;
               ELSE
                   #wykonuj_petle := false;
               END_IF;
           ELSE
               #wykonuj_petle := false;
           END_IF;
       END_WHILE;
       #wykonuj_petle := TRUE;
       #poz_temp := #hetman.pozycja;
       WHILE #wykonuj_petle DO
           #poz_temp.x -= 1;
           #poz_temp.y -= 1;
           IF "sprawdz_czy_na_szachownicy"(#poz_temp) = true THEN
               IF "sprawdz_czy_wolne"(pozycja := #poz_temp, szachownica := #szachownica) = true THEN
                   IF "sprawdz_czy_ruch_możliwy"(figura := #hetman, szachownica := #szachownica, pozycja := #poz_temp) = true  THEN
                       #hetman.mozliwe_ruchy[#indeks_mozliwych_ruchow] := #poz_temp;
                       #indeks_mozliwych_ruchow += 1;
                   END_IF;
               ELSIF "sprawdz_czy_zajete"(pozycja := #poz_temp, szachownica := #szachownica) = 1 THEN
                   IF "sprawdz_czy_ruch_możliwy"(figura := #hetman, szachownica := #szachownica, pozycja := #poz_temp) = true  THEN
                       #hetman.mozliwe_ruchy[#indeks_mozliwych_ruchow] := #poz_temp;
                       #indeks_mozliwych_ruchow += 1;
                       #wykonuj_petle := false;
                   END_IF;
               ELSE
                   #wykonuj_petle := false;
               END_IF;
           ELSE
               #wykonuj_petle := false;
           END_IF;
       END_WHILE;
       //ruch poziomo i pionowo
       #wykonuj_petle := TRUE;
       #poz_temp := #hetman.pozycja;
       WHILE #wykonuj_petle DO
           #poz_temp.x += 1;
           #poz_temp.y += 0;
           IF "sprawdz_czy_na_szachownicy"(#poz_temp) = true THEN
               IF "sprawdz_czy_wolne"(pozycja := #poz_temp, szachownica := #szachownica) = true THEN
                   IF "sprawdz_czy_ruch_możliwy"(figura := #hetman, szachownica := #szachownica, pozycja := #poz_temp) = true  THEN
                       #hetman.mozliwe_ruchy[#indeks_mozliwych_ruchow] := #poz_temp;
                       #indeks_mozliwych_ruchow += 1;
                   END_IF;
               ELSIF "sprawdz_czy_zajete"(pozycja := #poz_temp, szachownica := #szachownica) = 1 THEN
                   IF "sprawdz_czy_ruch_możliwy"(figura := #hetman, szachownica := #szachownica, pozycja := #poz_temp) = true  THEN
                       #hetman.mozliwe_ruchy[#indeks_mozliwych_ruchow] := #poz_temp;
                       #indeks_mozliwych_ruchow += 1;
                       #wykonuj_petle := false;
                   END_IF;
               ELSE
                   #wykonuj_petle := false;
               END_IF;
           ELSE
               #wykonuj_petle := false;
           END_IF;
       END_WHILE;
       #wykonuj_petle := TRUE;
       #poz_temp := #hetman.pozycja;
       WHILE #wykonuj_petle DO
           #poz_temp.x += 0;
           #poz_temp.y += 1;
           IF "sprawdz_czy_na_szachownicy"(#poz_temp) = true THEN
               IF "sprawdz_czy_wolne"(pozycja := #poz_temp, szachownica := #szachownica) = true THEN
                   IF "sprawdz_czy_ruch_możliwy"(figura := #hetman, szachownica := #szachownica, pozycja := #poz_temp) = true  THEN
                       #hetman.mozliwe_ruchy[#indeks_mozliwych_ruchow] := #poz_temp;
                       #indeks_mozliwych_ruchow += 1;
                   END_IF;
               ELSIF "sprawdz_czy_zajete"(pozycja := #poz_temp, szachownica := #szachownica) = 1 THEN
                   IF "sprawdz_czy_ruch_możliwy"(figura := #hetman, szachownica := #szachownica, pozycja := #poz_temp) = true  THEN
                       #hetman.mozliwe_ruchy[#indeks_mozliwych_ruchow] := #poz_temp;
                       #indeks_mozliwych_ruchow += 1;
                       #wykonuj_petle := false;
                   END_IF;
               ELSE
                   #wykonuj_petle := false;
               END_IF;
           ELSE
               #wykonuj_petle := false;
           END_IF;
       END_WHILE;
       #wykonuj_petle := TRUE;
       #poz_temp := #hetman.pozycja;
       WHILE #wykonuj_petle DO
           #poz_temp.x += -1;
           #poz_temp.y += 0;
           IF "sprawdz_czy_na_szachownicy"(#poz_temp) = true THEN
               IF "sprawdz_czy_wolne"(pozycja := #poz_temp, szachownica := #szachownica) = true THEN
                   IF "sprawdz_czy_ruch_możliwy"(figura := #hetman, szachownica := #szachownica, pozycja := #poz_temp) = true  THEN
                       #hetman.mozliwe_ruchy[#indeks_mozliwych_ruchow] := #poz_temp;
                       #indeks_mozliwych_ruchow += 1;
                   END_IF;
               ELSIF "sprawdz_czy_zajete"(pozycja := #poz_temp, szachownica := #szachownica) = 1 THEN
                   IF "sprawdz_czy_ruch_możliwy"(figura := #hetman, szachownica := #szachownica, pozycja := #poz_temp) = true  THEN
                       #hetman.mozliwe_ruchy[#indeks_mozliwych_ruchow] := #poz_temp;
                       #indeks_mozliwych_ruchow += 1;
                       #wykonuj_petle := false;
                   END_IF;
               ELSE
                   #wykonuj_petle := false;
               END_IF;
           ELSE
               #wykonuj_petle := false;
           END_IF;
       END_WHILE;
       #wykonuj_petle := TRUE;
       #poz_temp := #hetman.pozycja;
       WHILE #wykonuj_petle DO
           #poz_temp.x += 0;
           #poz_temp.y += -1;
           IF "sprawdz_czy_na_szachownicy"(#poz_temp) = true THEN
               IF "sprawdz_czy_wolne"(pozycja := #poz_temp, szachownica := #szachownica) = true THEN
                   IF "sprawdz_czy_ruch_możliwy"(figura := #hetman, szachownica := #szachownica, pozycja := #poz_temp) = true  THEN
                       #hetman.mozliwe_ruchy[#indeks_mozliwych_ruchow] := #poz_temp;
                       #indeks_mozliwych_ruchow += 1;
                   END_IF;
               ELSIF "sprawdz_czy_zajete"(pozycja := #poz_temp, szachownica := #szachownica) = 1 THEN
                   IF "sprawdz_czy_ruch_możliwy"(figura := #hetman, szachownica := #szachownica, pozycja := #poz_temp) = true  THEN
                       #hetman.mozliwe_ruchy[#indeks_mozliwych_ruchow] := #poz_temp;
                       #indeks_mozliwych_ruchow += 1;
                       #wykonuj_petle := false;
                   END_IF;
               ELSE
                   #wykonuj_petle := false;
               END_IF;
           ELSE
               #wykonuj_petle := false;
           END_IF;
       END_WHILE;


